(* CODESYS project experiment_with_CoDeSys_sp16.project
   Company: ifm electronic
   Description: Project template with CR711S configured 2.25MByte Standard 2.25MByte Safety
   Version: 2.4.15.0
   Title: ifmCR711S_TemplateProject

Project tree, tasks and I/O mapping:
  SafetyPLC : CR711S SIL2, ifm electronic, order no. CR711S, version 3.0.0.1
    application Application
      libraries: ifmR360-3, * (ifm electronic)
      task Task (cyclic, interval t#10ms, priority 1, watchdog t#8ms x 1) calls PLC_PRG
      global variables EVL
      program PLC_PRG [ST]
    Communication : Communication, ifm electronic, version 3.0.0.1
      CAN : CAN, ifm electronic, version 3.0.0.1
      Ethernet : Ethernet, ifm electronic, version 3.0.0.1
    HMI : HMI, ifm electronic, version 3.0.0.1
      User_LEDs : User_LEDs, ifm electronic, version 3.0.0.1
          input  UserLED0_I : LED_IEC_B_INPUT_MAPPING_TYPE  // UserLED0_I
          input  UserLED1_I : LED_IEC_B_INPUT_MAPPING_TYPE  // UserLED1_I
          input  UserLED2_I : LED_IEC_B_INPUT_MAPPING_TYPE  // UserLED2_I
          input  UserLED3_I : LED_IEC_B_INPUT_MAPPING_TYPE  // UserLED3_I
          output UserLED0_Q : LED_IEC_B_OUTPUT_MAPPING_TYPE  // User LED 0
          output UserLED1_Q : LED_IEC_B_OUTPUT_MAPPING_TYPE  // User LED 1
          output UserLED2_Q : LED_IEC_B_OUTPUT_MAPPING_TYPE  // User LED 2
          output UserLED3_Q : LED_IEC_B_OUTPUT_MAPPING_TYPE  // User LED 3
    Local_IO : Local_IO, ifm electronic, version 3.0.0.1
      Inputs : Inputs, ifm electronic, version 3.0.0.1
          input  IN0100_I : IN_MULTIFUNCTION_A_INPUT_MAPPING_TYPE  // IN0100_I
          input  IN0101_I : IN_MULTIFUNCTION_A_INPUT_MAPPING_TYPE  // IN0101_I
          input  IN0102_I : IN_MULTIFUNCTION_A_INPUT_MAPPING_TYPE  // IN0102_I
          input  IN0103_I : IN_MULTIFUNCTION_A_INPUT_MAPPING_TYPE  // IN0103_I
          input  IN0200_I : IN_MULTIFUNCTION_A_INPUT_MAPPING_TYPE  // IN0200_I
          input  IN0201_I : IN_MULTIFUNCTION_A_INPUT_MAPPING_TYPE  // IN0201_I
          input  IN0202_I : IN_MULTIFUNCTION_A_INPUT_MAPPING_TYPE  // IN0202_I
          input  IN0203_I : IN_MULTIFUNCTION_A_INPUT_MAPPING_TYPE  // IN0203_I
          input  IN0600_I : IN_MULTIFUNCTION_A_INPUT_MAPPING_TYPE  // IN0600_I
          input  IN0601_I : IN_MULTIFUNCTION_A_INPUT_MAPPING_TYPE  // IN0601_I
          input  IN0602_I : IN_MULTIFUNCTION_A_INPUT_MAPPING_TYPE  // IN0602_I
          input  IN0603_I : IN_MULTIFUNCTION_A_INPUT_MAPPING_TYPE  // IN0603_I
          input  IN0700_I : IN_MULTIFUNCTION_A_INPUT_MAPPING_TYPE  // IN0700_I
          input  IN0701_I : IN_MULTIFUNCTION_A_INPUT_MAPPING_TYPE  // IN0701_I
          input  IN0702_I : IN_MULTIFUNCTION_A_INPUT_MAPPING_TYPE  // IN0702_I
          input  IN0703_I : IN_MULTIFUNCTION_A_INPUT_MAPPING_TYPE  // IN0703_I
          input  IN0400_I : IN_RESISTOR_A_INPUT_MAPPING_TYPE  // IN0400_I
          input  IN0401_I : IN_RESISTOR_A_INPUT_MAPPING_TYPE  // IN0401_I
          input  IN0900_I : IN_RESISTOR_A_INPUT_MAPPING_TYPE  // IN0900_I
          input  IN0901_I : IN_RESISTOR_A_INPUT_MAPPING_TYPE  // IN0901_I
          input  IN0300_I : IN_DIGITAL_B_INPUT_MAPPING_TYPE  // IN0300_I
          input  IN0301_I : IN_DIGITAL_B_INPUT_MAPPING_TYPE  // IN0301_I
          input  IN0800_I : IN_DIGITAL_B_INPUT_MAPPING_TYPE  // IN0800_I
          input  IN0801_I : IN_DIGITAL_B_INPUT_MAPPING_TYPE  // IN0801_I
          input  COM_RESET_I : IN_COMMUNICATION_RESET_INPUT_MAPPING_TYPE  // COM_RESET_I
          input  IN0000_I : IN_FREQUENCY_B_CHANNEL_A_INPUT_MAPPING_TYPE  // IN0000_I
          input  IN0002_I : IN_FREQUENCY_B_CHANNEL_A_INPUT_MAPPING_TYPE  // IN0002_I
          input  IN0500_I : IN_FREQUENCY_B_CHANNEL_A_INPUT_MAPPING_TYPE  // IN0500_I
          input  IN0502_I : IN_FREQUENCY_B_CHANNEL_A_INPUT_MAPPING_TYPE  // IN0502_I
          input  IN0001_I : IN_FREQUENCY_B_CHANNEL_B_INPUT_MAPPING_TYPE  // IN0001_I
          input  IN0003_I : IN_FREQUENCY_B_CHANNEL_B_INPUT_MAPPING_TYPE  // IN0003_I
          input  IN0501_I : IN_FREQUENCY_B_CHANNEL_B_INPUT_MAPPING_TYPE  // IN0501_I
          input  IN0503_I : IN_FREQUENCY_B_CHANNEL_B_INPUT_MAPPING_TYPE  // IN0503_I
      Outputs : Outputs, ifm electronic, version 3.0.0.1
          input  OUT0006_I : OUT_PWM_40_BRIDGE_A_INPUT_MAPPING_TYPE  // OUT0006_I
          input  OUT0106_I : OUT_PWM_40_BRIDGE_A_INPUT_MAPPING_TYPE  // OUT0106_I
          input  OUT0206_I : OUT_PWM_40_BRIDGE_A_INPUT_MAPPING_TYPE  // OUT0206_I
          input  OUT0008_I : OUT_PWM_40_A_INPUT_MAPPING_TYPE  // OUT0008_I
          input  OUT0108_I : OUT_PWM_40_A_INPUT_MAPPING_TYPE  // OUT0108_I
          input  OUT0208_I : OUT_PWM_40_A_INPUT_MAPPING_TYPE  // OUT0208_I
          input  OUT0000_I : OUT_PWM_25_A_INPUT_MAPPING_TYPE  // OUT0000_I
          input  OUT0002_I : OUT_PWM_25_A_INPUT_MAPPING_TYPE  // OUT0002_I
          input  OUT0004_I : OUT_PWM_25_A_INPUT_MAPPING_TYPE  // OUT0004_I
          input  OUT0100_I : OUT_PWM_25_A_INPUT_MAPPING_TYPE  // OUT0100_I
          input  OUT0102_I : OUT_PWM_25_A_INPUT_MAPPING_TYPE  // OUT0102_I
          input  OUT0104_I : OUT_PWM_25_A_INPUT_MAPPING_TYPE  // OUT0104_I
          input  OUT0200_I : OUT_PWM_25_A_INPUT_MAPPING_TYPE  // OUT0200_I
          input  OUT0202_I : OUT_PWM_25_A_INPUT_MAPPING_TYPE  // OUT0202_I
          input  OUT0204_I : OUT_PWM_25_A_INPUT_MAPPING_TYPE  // OUT0204_I
          input  OUT3001_I : OUT_VOLTAGE_A_INPUT_MAPPING_TYPE  // OUT3001_I
          input  OUT3000_I : OUT_SUPPLY_A_INPUT_MAPPING_TYPE  // OUT3000_I
          input  OUT0001_I : OUT_PWM_25_B_INPUT_MAPPING_TYPE  // OUT0001_I
          input  OUT0003_I : OUT_PWM_25_B_INPUT_MAPPING_TYPE  // OUT0003_I
          input  OUT0005_I : OUT_PWM_25_B_INPUT_MAPPING_TYPE  // OUT0005_I
          input  OUT0101_I : OUT_PWM_25_B_INPUT_MAPPING_TYPE  // OUT0101_I
          input  OUT0103_I : OUT_PWM_25_B_INPUT_MAPPING_TYPE  // OUT0103_I
          input  OUT0105_I : OUT_PWM_25_B_INPUT_MAPPING_TYPE  // OUT0105_I
          input  OUT0201_I : OUT_PWM_25_B_INPUT_MAPPING_TYPE  // OUT0201_I
          input  OUT0203_I : OUT_PWM_25_B_INPUT_MAPPING_TYPE  // OUT0203_I
          input  OUT0205_I : OUT_PWM_25_B_INPUT_MAPPING_TYPE  // OUT0205_I
          input  OUT0007_I : OUT_PWM_40_BRIDGE_A_INPUT_MAPPING_TYPE  // OUT0007_I
          input  OUT0107_I : OUT_PWM_40_BRIDGE_A_INPUT_MAPPING_TYPE  // OUT0107_I
          input  OUT0207_I : OUT_PWM_40_BRIDGE_A_INPUT_MAPPING_TYPE  // OUT0207_I
          output OUT0006_Q : OUT_PWM_40_BRIDGE_A_OUTPUT_MAPPING_TYPE  // OUT0006_Q
          output OUT0106_Q : OUT_PWM_40_BRIDGE_A_OUTPUT_MAPPING_TYPE  // OUT0106_Q
          output OUT0206_Q : OUT_PWM_40_BRIDGE_A_OUTPUT_MAPPING_TYPE  // OUT0206_Q
          output OUT0008_Q : OUT_PWM_40_A_OUTPUT_MAPPING_TYPE  // OUT0008_Q
          output OUT0108_Q : OUT_PWM_40_A_OUTPUT_MAPPING_TYPE  // OUT0108_Q
          output OUT0208_Q : OUT_PWM_40_A_OUTPUT_MAPPING_TYPE  // OUT0208_Q
          output OUT0000_Q : OUT_PWM_25_A_OUTPUT_MAPPING_TYPE  // OUT0000_Q
          output OUT0002_Q : OUT_PWM_25_A_OUTPUT_MAPPING_TYPE  // OUT0002_Q
          output OUT0004_Q : OUT_PWM_25_A_OUTPUT_MAPPING_TYPE  // OUT0004_Q
          output OUT0100_Q : OUT_PWM_25_A_OUTPUT_MAPPING_TYPE  // OUT0100_Q
          output OUT0102_Q : OUT_PWM_25_A_OUTPUT_MAPPING_TYPE  // OUT0102_Q
          output OUT0104_Q : OUT_PWM_25_A_OUTPUT_MAPPING_TYPE  // OUT0104_Q
          output OUT0200_Q : OUT_PWM_25_A_OUTPUT_MAPPING_TYPE  // OUT0200_Q
          output OUT0202_Q : OUT_PWM_25_A_OUTPUT_MAPPING_TYPE  // OUT0202_Q
          output OUT0204_Q : OUT_PWM_25_A_OUTPUT_MAPPING_TYPE  // OUT0204_Q
          output OUT3001_Q : OUT_VOLTAGE_A_OUTPUT_MAPPING_TYPE  // OUT3001_Q
          output OUT3000_Q : OUT_SUPPLY_A_OUTPUT_MAPPING_TYPE  // OUT3000_Q
          output OUT0001_Q : OUT_PWM_25_B_OUTPUT_MAPPING_TYPE  // OUT0001_Q
          output OUT0003_Q : OUT_PWM_25_B_OUTPUT_MAPPING_TYPE  // OUT0003_Q
          output OUT0005_Q : OUT_PWM_25_B_OUTPUT_MAPPING_TYPE  // OUT0005_Q
          output OUT0101_Q : OUT_PWM_25_B_OUTPUT_MAPPING_TYPE  // OUT0101_Q
          output OUT0103_Q : OUT_PWM_25_B_OUTPUT_MAPPING_TYPE  // OUT0103_Q
          output OUT0105_Q : OUT_PWM_25_B_OUTPUT_MAPPING_TYPE  // OUT0105_Q
          output OUT0201_Q : OUT_PWM_25_B_OUTPUT_MAPPING_TYPE  // OUT0201_Q
          output OUT0203_Q : OUT_PWM_25_B_OUTPUT_MAPPING_TYPE  // OUT0203_Q
          output OUT0205_Q : OUT_PWM_25_B_OUTPUT_MAPPING_TYPE  // OUT0205_Q
          output OUT0007_Q : OUT_PWM_40_BRIDGE_A_OUTPUT_MAPPING_TYPE  // OUT0007_Q
          output OUT0107_Q : OUT_PWM_40_BRIDGE_A_OUTPUT_MAPPING_TYPE  // OUT0107_Q
          output OUT0207_Q : OUT_PWM_40_BRIDGE_A_OUTPUT_MAPPING_TYPE  // OUT0207_Q
      System_Inputs : System_Inputs, ifm electronic, version 3.0.0.1
          input  VBB30 : IN_SYSTEM_VOLTAGE_INPUT_MAPPING_TYPE  // VBB30
          input  VBB15 : IN_SYSTEM_VOLTAGE_INPUT_MAPPING_TYPE  // VBB15
          input  TemperatureBoard0 : IN_TEMPERATURE_INPUT_MAPPING_TYPE  // TemperatureBoard0
          input  TemperatureChip0 : IN_TEMPERATURE_INPUT_MAPPING_TYPE  // TemperatureChip0
      System_Outputs : System_Outputs, ifm electronic, version 3.0.0.1
          input  VBB0_SW_I : OUT_GROUP_SWITCH_INPUT_MAPPING_TYPE  // VBB0_SW_I
          input  VBB1_SW_I : OUT_GROUP_SWITCH_INPUT_MAPPING_TYPE  // VBB1_SW_I
          input  VBB2_SW_I : OUT_GROUP_SWITCH_INPUT_MAPPING_TYPE  // VBB2_SW_I
          output VBB0_SW_Q : OUT_GROUP_SWITCH_OUTPUT_MAPPING_TYPE  // VBB0_SW_Q
          output VBB1_SW_Q : OUT_GROUP_SWITCH_OUTPUT_MAPPING_TYPE  // VBB1_SW_Q
          output VBB2_SW_Q : OUT_GROUP_SWITCH_OUTPUT_MAPPING_TYPE  // VBB2_SW_Q
          output SUPPLY_SWITCH_Q : OUT_SYS_SWITCH_OUTPUT_MAPPING_TYPE  // SUPPLY_SWITCH_Q
  StandardPLC : CR711S Standard, ifm electronic, order no. CR711S, version 3.0.0.1
    application Application
      libraries: ifmR360-3, * (ifm electronic); SysTime, 3.5.9.0 (System); 3S CANopenStack, 3.5.11.0 (3S - Smart Software Solutions GmbH); CAA CiA 405, 3.5.8.0 (CAA Technical Workgroup); Converted Hydraulic library, 0.0.0.1 (ifmWT); StringUtils, 3.5.15.0 (System); SysCom, 3.5.15.0 (System); SysMem23, 3.5.13.0 (System); TD3-1 Framework, 3.1.0.1 (Ojjo); Util, * (System); Motor3-1 control, 3.1.0.1 (Ojjo); Standard, * (System); VisuDialogs, * (System)
      task Task (cyclic, interval 20 ms, priority 1) calls PLC_PRG
      EVC
      GlobalVars/
        global variables Test1Vars
        global variables Test2Vars
        global variables Dims
        global variables Positions
        global variables GPS_Data
        global variables Ojjo_TD
      POUs/
        program PLC_PRG [ST]
        function block ConvertDiag [ST]
        function ConvDiag [ST]
        program Type_conversions [ST]
        function Checksum [ST]
        function Checksum_wLength [ST]
        function IsExtendedCAN [ST]
        function block getElapsedTime [ST]
        Utilities/
          function MemBlockLength [ST]
          Conversions/
            function pSQR [ST]
            function SqrReals [ST]
            function AsciiToReal [ST]
            function ArrayOfBytesToLWORD [ST]
            function ConvLWORDtoDecimal [ST]
            function block REAL_TO_BYTE_ARRAY [ST]
            function ArrayOfUsintsToLWORD [ST]
            function ATAN_DEG [ST]
            function COS_DEG [ST]
            function SIN_DEG [ST]
            function TAN_DEG [ST]
            function CanMsgIdToNodeIndexSubIndex [ST]
            function CanNodeIndexSubIndexToJ1939MsgId [ST]
            function ACOS_DEG [ST]
            function ASIN_DEG [ST]
            function ByteArrayToText [ST]
            function ddt [ST]
            function ddt_max [ST]
            function block ddt_layers [ST]
          ProfileGen/
            function ProfileGenerator_2d [ST]
            function CurveGenerator_2d [ST]
            data type CurveTypes
            function SetpointInit [ST]
            TDcontrolCode/
              function setVelAccel [ST]
              data type sSetpoint
              function POS_ENGR_TO_RAW [ST]
              data type sFeedback
              function FeedbackInit [ST]
              function VEL_ENGR_TO_RAW [ST]
            function block ScurveProfiler [ST]
            function AutotargetIncrementPos [ST]
            function GpsFeedbackAutotarget [ST]
            function TrapezoidStart [ST]
            function TrapezoidStart_jerk [ST]
          function block DataSmoothing [ST]
          function block DataSmoothing_1 [ST]
          function block DataSmoothing_2 [ST]
          function UpperBoundBool [ST]
        GPS/
          data type eScrewParameters
          function RotateGpsTdToWorldNS [ST]
          data type eGPS
          data type eGpsDataCategories
          function GpsTdToWorldFixedYaw [ST]
          function GPS_Y_TO_BS_ANGLE [ST]
          function GPS_Y_TO_BS_ANGLE_1 [ST]
          function GPS_Y_TO_BS_ANGLE_2 [ST]
          function GpsTransform3d [ST]
          function GpsAutotargetInRange [ST]
          data type sGPSaxis
          function block GpsUpdate [ST]
          function block GPS [ST]
          program CheckGpsInRange [ST]
          function TD_SIM [ST]
          function GpsTdToWorldFixAll2d [ST]
          program GpsAutoTrack_1 [ST]
          function GpsAutoTrack [ST]
          function GpsAxisIsNearTarget [ST]
          function GpsAxisIsOnTarget [ST]
          function DecodePnezD [ST]
        Test_PRGs/
          program pnezD_decoding [ST]
          program DynamicList [ST]
          program Arrays [ST]
          program Parsing [ST]
      Network Variables/
        global variables PLC_TRANSMIT_1
      DUTs/
        data type color
        data type SqrStruct
        data type Diag
        data type Coordinates2d
        data type Coordinates3d
        data type sScrewParams
      Visualizations/
        visualisation GPS_RANGE
        visualisation FUNCTION_CHECK
        visualisation P_GPS_testing
        visualisation GRAPH_FUNCTION_RESULTS
    Communication : Communication, ifm electronic, version 3.0.0.1
      CAN : CAN, ifm electronic, version 3.0.0.1
        CANbus_3 : CANbus, ifm electronic, version 1.0.0.0
            settings: NetID = 3
          J1939_Manager : J1939_Manager, 3S - Smart Software Solutions GmbH, version 3.5.10.0
            Rx_KARTECH : J1939_ECU, 3S - Smart Software Solutions GmbH, version 3.5.9.0
                settings: NAME = 16#1060000000000000; Communication Watchdog Timeout Period = 16#05DC ms; Activated PGs = 0; PG Offline Data.Name = "Group0"; PG Offline Data.Description = ""; PG Online Data.PGN = 65280; PG Online Data.Length (Bytes) = 8; PG Transmission Settings.Destination Address = 255; PG Transmission Settings.CycleTimeFactor = 1; Signal Offline Data.SPN = 0; Signal Offline Data.Name = "Toggle"; Signal Offline Data.Description = ""; Signal Offline Data.Unit = ""; Signal Offline Data.Min = 0; Signal Offline Data.Max = 0; Signal Online Data.BitSize = 1; Signal Online Data.BitPosition = 0; Convert Data.Flags = 3; Convert Data.pSigValue = 0; Convert Data.Scaling = 4607182418800017408; Convert Data.Offset = 0; Signal Offline Data.SPN = 0; Signal Offline Data.Name = "rf_CANlink"; Signal Offline Data.Description = ""; Signal Offline Data.Unit = ""; Signal Offline Data.Min = 0; Signal Offline Data.Max = 0; Signal Online Data.BitSize = 1; Signal Online Data.BitPosition = 1; Convert Data.Flags = 3; Convert Data.pSigValue = 0; Convert Data.Scaling = 4607182418800017408; Convert Data.Offset = 0; Signal Offline Data.SPN = 0; Signal Offline Data.Name = "DI1"; Signal Offline Data.Description = ""; Signal Offline Data.Unit = ""; Signal Offline Data.Min = 0; Signal Offline Data.Max = 0; Signal Online Data.BitSize = 1;
                  Signal Online Data.BitPosition = 16; Convert Data.Flags = 3; Convert Data.pSigValue = 0; Convert Data.Scaling = 4607182418800017408; Convert Data.Offset = 0; Signal Offline Data.SPN = 0; Signal Offline Data.Name = "DI2"; Signal Offline Data.Description = ""; Signal Offline Data.Unit = ""; Signal Offline Data.Min = 0; Signal Offline Data.Max = 0; Signal Online Data.BitSize = 1; Signal Online Data.BitPosition = 17; Convert Data.Flags = 3; Convert Data.pSigValue = 0; Convert Data.Scaling = 4607182418800017408; Convert Data.Offset = 0; Signal Offline Data.SPN = 0; Signal Offline Data.Name = "DI3"; Signal Offline Data.Description = ""; Signal Offline Data.Unit = ""; Signal Offline Data.Min = 0; Signal Offline Data.Max = 0; Signal Online Data.BitSize = 1; Signal Online Data.BitPosition = 18; Convert Data.Flags = 3; Convert Data.pSigValue = 0; Convert Data.Scaling = 4607182418800017408; Convert Data.Offset = 0; Signal Offline Data.SPN = 0; Signal Offline Data.Name = "DI4"; Signal Offline Data.Description = ""; Signal Offline Data.Unit = ""; Signal Offline Data.Min = 0; Signal Offline Data.Max = 0; Signal Online Data.BitSize = 1; Signal Online Data.BitPosition = 19; Convert Data.Flags = 3; Convert Data.pSigValue = 0; Convert Data.Scaling = 4607182418800017408;
                  Convert Data.Offset = 0; Signal Offline Data.SPN = 0; Signal Offline Data.Name = "DI5"; Signal Offline Data.Description = ""; Signal Offline Data.Unit = ""; Signal Offline Data.Min = 0; Signal Offline Data.Max = 0; Signal Online Data.BitSize = 1; Signal Online Data.BitPosition = 20; Convert Data.Flags = 3; Convert Data.pSigValue = 0; Convert Data.Scaling = 4607182418800017408; Convert Data.Offset = 0; Signal Offline Data.SPN = 0; Signal Offline Data.Name = "DI6"; Signal Offline Data.Description = ""; Signal Offline Data.Unit = ""; Signal Offline Data.Min = 0; Signal Offline Data.Max = 0; Signal Online Data.BitSize = 1; Signal Online Data.BitPosition = 21; Convert Data.Flags = 3; Convert Data.pSigValue = 0; Convert Data.Scaling = 4607182418800017408; Convert Data.Offset = 0; Signal Offline Data.SPN = 0; Signal Offline Data.Name = "DI7"; Signal Offline Data.Description = ""; Signal Offline Data.Unit = ""; Signal Offline Data.Min = 0; Signal Offline Data.Max = 0; Signal Online Data.BitSize = 1; Signal Online Data.BitPosition = 22; Convert Data.Flags = 3; Convert Data.pSigValue = 0; Convert Data.Scaling = 4607182418800017408; Convert Data.Offset = 0; Signal Offline Data.SPN = 0; Signal Offline Data.Name = "DI8"; Signal Offline Data.Description = "";
                  Signal Offline Data.Unit = ""; Signal Offline Data.Min = 0; Signal Offline Data.Max = 0; Signal Online Data.BitSize = 1; Signal Online Data.BitPosition = 23; Convert Data.Flags = 3; Convert Data.pSigValue = 0; Convert Data.Scaling = 4607182418800017408; Convert Data.Offset = 0; Signal Offline Data.SPN = 0; Signal Offline Data.Name = "DI9"; Signal Offline Data.Description = ""; Signal Offline Data.Unit = ""; Signal Offline Data.Min = 0; Signal Offline Data.Max = 0; Signal Online Data.BitSize = 1; Signal Online Data.BitPosition = 24; Convert Data.Flags = 3; Convert Data.pSigValue = 0; Convert Data.Scaling = 4607182418800017408; Convert Data.Offset = 0; Signal Offline Data.SPN = 0; Signal Offline Data.Name = "DI10"; Signal Offline Data.Description = ""; Signal Offline Data.Unit = ""; Signal Offline Data.Min = 0; Signal Offline Data.Max = 0; Signal Online Data.BitSize = 1; Signal Online Data.BitPosition = 25; Convert Data.Flags = 3; Convert Data.pSigValue = 0; Convert Data.Scaling = 4607182418800017408; Convert Data.Offset = 0; Signal Offline Data.SPN = 0; Signal Offline Data.Name = "DI11"; Signal Offline Data.Description = ""; Signal Offline Data.Unit = ""; Signal Offline Data.Min = 0; Signal Offline Data.Max = 0; Signal Online Data.BitSize = 1;
                  Signal Online Data.BitPosition = 26; Convert Data.Flags = 3; Convert Data.pSigValue = 0; Convert Data.Scaling = 4607182418800017408; Convert Data.Offset = 0; Signal Offline Data.SPN = 0; Signal Offline Data.Name = "DI12"; Signal Offline Data.Description = ""; Signal Offline Data.Unit = ""; Signal Offline Data.Min = 0; Signal Offline Data.Max = 0; Signal Online Data.BitSize = 1; Signal Online Data.BitPosition = 27; Convert Data.Flags = 3; Convert Data.pSigValue = 0; Convert Data.Scaling = 4607182418800017408; Convert Data.Offset = 0; Signal Offline Data.SPN = 0; Signal Offline Data.Name = "DI13"; Signal Offline Data.Description = ""; Signal Offline Data.Unit = ""; Signal Offline Data.Min = 0; Signal Offline Data.Max = 0; Signal Online Data.BitSize = 1; Signal Online Data.BitPosition = 28; Convert Data.Flags = 3; Convert Data.pSigValue = 0; Convert Data.Scaling = 4607182418800017408; Convert Data.Offset = 0; Signal Offline Data.SPN = 0; Signal Offline Data.Name = "DI14"; Signal Offline Data.Description = ""; Signal Offline Data.Unit = ""; Signal Offline Data.Min = 0; Signal Offline Data.Max = 0; Signal Online Data.BitSize = 1; Signal Online Data.BitPosition = 29; Convert Data.Flags = 3; Convert Data.pSigValue = 0; Convert Data.Scaling = 4607182418800017408;
                  Convert Data.Offset = 0; Signal Offline Data.SPN = 0; Signal Offline Data.Name = "DI15"; Signal Offline Data.Description = ""; Signal Offline Data.Unit = ""; Signal Offline Data.Min = 0; Signal Offline Data.Max = 0; Signal Online Data.BitSize = 1; Signal Online Data.BitPosition = 30; Convert Data.Flags = 3; Convert Data.pSigValue = 0; Convert Data.Scaling = 4607182418800017408; Convert Data.Offset = 0; Signal Offline Data.SPN = 0; Signal Offline Data.Name = "DI16"; Signal Offline Data.Description = ""; Signal Offline Data.Unit = ""; Signal Offline Data.Min = 0; Signal Offline Data.Max = 0; Signal Online Data.BitSize = 1; Signal Online Data.BitPosition = 31; Convert Data.Flags = 3; Convert Data.pSigValue = 0; Convert Data.Scaling = 4607182418800017408; Convert Data.Offset = 0; Signal Offline Data.SPN = 0; Signal Offline Data.Name = "DI17"; Signal Offline Data.Description = ""; Signal Offline Data.Unit = ""; Signal Offline Data.Min = 0; Signal Offline Data.Max = 0; Signal Online Data.BitSize = 1; Signal Online Data.BitPosition = 32; Convert Data.Flags = 3; Convert Data.pSigValue = 0; Convert Data.Scaling = 4607182418800017408; Convert Data.Offset = 0; Signal Offline Data.SPN = 0; Signal Offline Data.Name = "DI18"; Signal Offline Data.Description = "";
                  Signal Offline Data.Unit = ""; Signal Offline Data.Min = 0; Signal Offline Data.Max = 0; Signal Online Data.BitSize = 1; Signal Online Data.BitPosition = 33; Convert Data.Flags = 3; Convert Data.pSigValue = 0; Convert Data.Scaling = 4607182418800017408; Convert Data.Offset = 0; Signal Offline Data.SPN = 0; Signal Offline Data.Name = "DI19"; Signal Offline Data.Description = ""; Signal Offline Data.Unit = ""; Signal Offline Data.Min = 0; Signal Offline Data.Max = 0; Signal Online Data.BitSize = 1; Signal Online Data.BitPosition = 34; Convert Data.Flags = 3; Convert Data.pSigValue = 0; Convert Data.Scaling = 4607182418800017408; Convert Data.Offset = 0; Signal Offline Data.SPN = 0; Signal Offline Data.Name = "DI20"; Signal Offline Data.Description = ""; Signal Offline Data.Unit = ""; Signal Offline Data.Min = 0; Signal Offline Data.Max = 0; Signal Online Data.BitSize = 1; Signal Online Data.BitPosition = 35; Convert Data.Flags = 3; Convert Data.pSigValue = 0; Convert Data.Scaling = 4607182418800017408; Convert Data.Offset = 0; PG Offline Data.Name = "Group1"; PG Offline Data.Description = ""; PG Online Data.PGN = 65281; PG Online Data.Length (Bytes) = 8; PG Transmission Settings.Destination Address = 255; PG Transmission Settings.CycleTimeFactor = 1; Signal Offline Data.SPN = 0;
                  Signal Offline Data.Name = "AI1"; Signal Offline Data.Description = ""; Signal Offline Data.Unit = ""; Signal Offline Data.Min = 0; Signal Offline Data.Max = 0; Signal Online Data.BitSize = 8; Signal Online Data.BitPosition = 0; Convert Data.Flags = 3; Convert Data.pSigValue = 0; Convert Data.Scaling = 4607182418800017408; Convert Data.Offset = 0; Signal Offline Data.SPN = 0; Signal Offline Data.Name = "AI2"; Signal Offline Data.Description = ""; Signal Offline Data.Unit = ""; Signal Offline Data.Min = 0; Signal Offline Data.Max = 0; Signal Online Data.BitSize = 8; Signal Online Data.BitPosition = 8; Convert Data.Flags = 3; Convert Data.pSigValue = 0; Convert Data.Scaling = 4607182418800017408; Convert Data.Offset = 0; Signal Offline Data.SPN = 0; Signal Offline Data.Name = "AI3"; Signal Offline Data.Description = ""; Signal Offline Data.Unit = ""; Signal Offline Data.Min = 0; Signal Offline Data.Max = 0; Signal Online Data.BitSize = 8; Signal Online Data.BitPosition = 16; Convert Data.Flags = 3; Convert Data.pSigValue = 0; Convert Data.Scaling = 4607182418800017408; Convert Data.Offset = 0; Signal Offline Data.SPN = 0; Signal Offline Data.Name = "AI4"; Signal Offline Data.Description = ""; Signal Offline Data.Unit = ""; Signal Offline Data.Min = 0;
                  Signal Offline Data.Max = 0; Signal Online Data.BitSize = 8; Signal Online Data.BitPosition = 24; Convert Data.Flags = 3; Convert Data.pSigValue = 0; Convert Data.Scaling = 4607182418800017408; Convert Data.Offset = 0; Signal Offline Data.SPN = 0; Signal Offline Data.Name = "AI5"; Signal Offline Data.Description = ""; Signal Offline Data.Unit = ""; Signal Offline Data.Min = 0; Signal Offline Data.Max = 0; Signal Online Data.BitSize = 8; Signal Online Data.BitPosition = 32; Convert Data.Flags = 3; Convert Data.pSigValue = 0; Convert Data.Scaling = 4607182418800017408; Convert Data.Offset = 0; Signal Offline Data.SPN = 0; Signal Offline Data.Name = "AI6"; Signal Offline Data.Description = ""; Signal Offline Data.Unit = ""; Signal Offline Data.Min = 0; Signal Offline Data.Max = 0; Signal Online Data.BitSize = 8; Signal Online Data.BitPosition = 40; Convert Data.Flags = 3; Convert Data.pSigValue = 0; Convert Data.Scaling = 4607182418800017408; Convert Data.Offset = 0; Signal Offline Data.SPN = 0; Signal Offline Data.Name = "AI7"; Signal Offline Data.Description = ""; Signal Offline Data.Unit = ""; Signal Offline Data.Min = 0; Signal Offline Data.Max = 0; Signal Online Data.BitSize = 8; Signal Online Data.BitPosition = 48; Convert Data.Flags = 3;
                  Convert Data.pSigValue = 0; Convert Data.Scaling = 4607182418800017408; Convert Data.Offset = 0; Signal Offline Data.SPN = 0; Signal Offline Data.Name = "AI8"; Signal Offline Data.Description = ""; Signal Offline Data.Unit = ""; Signal Offline Data.Min = 0; Signal Offline Data.Max = 0; Signal Online Data.BitSize = 8; Signal Online Data.BitPosition = 56; Convert Data.Flags = 3; Convert Data.pSigValue = 0; Convert Data.Scaling = 4607182418800017408; Convert Data.Offset = 0; PG Offline Data.Name = "Group2"; PG Offline Data.Description = ""; PG Online Data.PGN = 65282; PG Online Data.Length (Bytes) = 8; PG Transmission Settings.Destination Address = 255; PG Transmission Settings.CycleTimeFactor = 1; Signal Offline Data.SPN = 0; Signal Offline Data.Name = "BatteryVoltage"; Signal Offline Data.Description = ""; Signal Offline Data.Unit = ""; Signal Offline Data.Min = 0; Signal Offline Data.Max = 0; Signal Online Data.BitSize = 16; Signal Online Data.BitPosition = 0; Convert Data.Flags = 3; Convert Data.pSigValue = 0; Convert Data.Scaling = 4607182418800017408; Convert Data.Offset = 4587366580439587226; Signal Offline Data.SPN = 0; Signal Offline Data.Name = "low_voltage"; Signal Offline Data.Description = ""; Signal Offline Data.Unit = ""; Signal Offline Data.Min = 0; Signal Offline Data.Max = 0; Signal Online Data.BitSize = 1;
                  Signal Online Data.BitPosition = 16; Convert Data.Flags = 3; Convert Data.pSigValue = 0; Convert Data.Scaling = 4607182418800017408; Convert Data.Offset = 0; Signal Offline Data.SPN = 0; Signal Offline Data.Name = "aiInput1err"; Signal Offline Data.Description = ""; Signal Offline Data.Unit = ""; Signal Offline Data.Min = 0; Signal Offline Data.Max = 0; Signal Online Data.BitSize = 1; Signal Online Data.BitPosition = 17; Convert Data.Flags = 3; Convert Data.pSigValue = 0; Convert Data.Scaling = 4607182418800017408; Convert Data.Offset = 0; Signal Offline Data.SPN = 0; Signal Offline Data.Name = "aiInput2err"; Signal Offline Data.Description = ""; Signal Offline Data.Unit = ""; Signal Offline Data.Min = 0; Signal Offline Data.Max = 0; Signal Online Data.BitSize = 1; Signal Online Data.BitPosition = 18; Convert Data.Flags = 3; Convert Data.pSigValue = 0; Convert Data.Scaling = 4607182418800017408; Convert Data.Offset = 0; Signal Offline Data.SPN = 0; Signal Offline Data.Name = "aiInput3err"; Signal Offline Data.Description = ""; Signal Offline Data.Unit = ""; Signal Offline Data.Min = 0; Signal Offline Data.Max = 0; Signal Online Data.BitSize = 1; Signal Online Data.BitPosition = 19; Convert Data.Flags = 3; Convert Data.pSigValue = 0; Convert Data.Scaling = 4607182418800017408;
                  Convert Data.Offset = 0; Signal Offline Data.SPN = 0; Signal Offline Data.Name = "aiInput4err"; Signal Offline Data.Description = ""; Signal Offline Data.Unit = ""; Signal Offline Data.Min = 0; Signal Offline Data.Max = 0; Signal Online Data.BitSize = 1; Signal Online Data.BitPosition = 20; Convert Data.Flags = 3; Convert Data.pSigValue = 0; Convert Data.Scaling = 4607182418800017408; Convert Data.Offset = 0; Signal Offline Data.SPN = 0; Signal Offline Data.Name = "aiInput5err"; Signal Offline Data.Description = ""; Signal Offline Data.Unit = ""; Signal Offline Data.Min = 0; Signal Offline Data.Max = 0; Signal Online Data.BitSize = 1; Signal Online Data.BitPosition = 21; Convert Data.Flags = 3; Convert Data.pSigValue = 0; Convert Data.Scaling = 4607182418800017408; Convert Data.Offset = 0; Signal Offline Data.SPN = 0; Signal Offline Data.Name = "aiInput6err"; Signal Offline Data.Description = ""; Signal Offline Data.Unit = ""; Signal Offline Data.Min = 0; Signal Offline Data.Max = 0; Signal Online Data.BitSize = 1; Signal Online Data.BitPosition = 22; Convert Data.Flags = 3; Convert Data.pSigValue = 0; Convert Data.Scaling = 4607182418800017408; Convert Data.Offset = 0; Signal Offline Data.SPN = 0; Signal Offline Data.Name = "aiInput7err"; Signal Offline Data.Description = "";
                  Signal Offline Data.Unit = ""; Signal Offline Data.Min = 0; Signal Offline Data.Max = 0; Signal Online Data.BitSize = 1; Signal Online Data.BitPosition = 23; Convert Data.Flags = 3; Convert Data.pSigValue = 0; Convert Data.Scaling = 4607182418800017408; Convert Data.Offset = 0; Signal Offline Data.SPN = 0; Signal Offline Data.Name = "aiInput8err"; Signal Offline Data.Description = ""; Signal Offline Data.Unit = ""; Signal Offline Data.Min = 0; Signal Offline Data.Max = 0; Signal Online Data.BitSize = 1; Signal Online Data.BitPosition = 24; Convert Data.Flags = 3; Convert Data.pSigValue = 0; Convert Data.Scaling = 4607182418800017408; Convert Data.Offset = 0; Signal Offline Data.SPN = 0; Signal Offline Data.Name = "VendorID"; Signal Offline Data.Description = ""; Signal Offline Data.Unit = ""; Signal Offline Data.Min = 0; Signal Offline Data.Max = 0; Signal Online Data.BitSize = 7; Signal Online Data.BitPosition = 25; Convert Data.Flags = 3; Convert Data.pSigValue = 0; Convert Data.Scaling = 4607182418800017408; Convert Data.Offset = 0; Signal Offline Data.SPN = 0; Signal Offline Data.Name = "Byte3"; Signal Offline Data.Description = ""; Signal Offline Data.Unit = ""; Signal Offline Data.Min = 0; Signal Offline Data.Max = 0; Signal Online Data.BitSize = 8;
                  Signal Online Data.BitPosition = 32; Convert Data.Flags = 3; Convert Data.pSigValue = 0; Convert Data.Scaling = 4607182418800017408; Convert Data.Offset = 0; Signal Offline Data.SPN = 0; Signal Offline Data.Name = "Byte4"; Signal Offline Data.Description = ""; Signal Offline Data.Unit = ""; Signal Offline Data.Min = 0; Signal Offline Data.Max = 0; Signal Online Data.BitSize = 8; Signal Online Data.BitPosition = 40; Convert Data.Flags = 3; Convert Data.pSigValue = 0; Convert Data.Scaling = 4607182418800017408; Convert Data.Offset = 0; Signal Offline Data.SPN = 0; Signal Offline Data.Name = "Byte5"; Signal Offline Data.Description = ""; Signal Offline Data.Unit = ""; Signal Offline Data.Min = 0; Signal Offline Data.Max = 0; Signal Online Data.BitSize = 8; Signal Online Data.BitPosition = 48; Convert Data.Flags = 3; Convert Data.pSigValue = 0; Convert Data.Scaling = 4607182418800017408; Convert Data.Offset = 0; Signal Offline Data.SPN = 0; Signal Offline Data.Name = "Byte6"; Signal Offline Data.Description = ""; Signal Offline Data.Unit = ""; Signal Offline Data.Min = 0; Signal Offline Data.Max = 0; Signal Online Data.BitSize = 8; Signal Online Data.BitPosition = 56; Convert Data.Flags = 3; Convert Data.pSigValue = 0; Convert Data.Scaling = 4607182418800017408;
                  Convert Data.Offset = 0; Signal Offline Data.SPN = 0; Signal Offline Data.Name = "Byte7"; Signal Offline Data.Description = ""; Signal Offline Data.Unit = ""; Signal Offline Data.Min = 0; Signal Offline Data.Max = 0; Signal Online Data.BitSize = 8; Signal Online Data.BitPosition = 57; Convert Data.Flags = 3; Convert Data.pSigValue = 0; Convert Data.Scaling = 4607182418800017408; Convert Data.Offset = 0; Activated PGs = 0
            LHP_Telematics : J1939_ECU, 3S - Smart Software Solutions GmbH, version 3.5.9.0
                settings: NAME = 16#0000000000000000; Communication Watchdog Timeout Period = 16#05DC ms; Activated PGs = 3; PG Offline Data.Name = "VP"; PG Offline Data.Description = "Vehicle Position"; PG Online Data.PGN = 65267; PG Online Data.Length (Bytes) = 8; PG Transmission Settings.Destination Address = 255; PG Transmission Settings.CycleTimeFactor = 1; Signal Offline Data.SPN = 584; Signal Offline Data.Name = "Latitude"; Signal Offline Data.Description = "Latitude position of the vehicle."; Signal Offline Data.Unit = "deg"; Signal Offline Data.Min = -210; Signal Offline Data.Max = 211.1008122; Signal Online Data.BitSize = 32; Signal Online Data.BitPosition = 0; Convert Data.Flags = 3; Convert Data.pSigValue = 0; Convert Data.Scaling = 4502148214488346440; Convert Data.Offset = 13864964771557670912; Signal Offline Data.SPN = 585; Signal Offline Data.Name = "Longitude"; Signal Offline Data.Description = "Longitude position of the vehicle."; Signal Offline Data.Unit = "deg"; Signal Offline Data.Min = -210; Signal Offline Data.Max = 211.1008122; Signal Online Data.BitSize = 32; Signal Online Data.BitPosition = 32; Convert Data.Flags = 3; Convert Data.pSigValue = 0; Convert Data.Scaling = 4502148214488346440; Convert Data.Offset = 13864964771557670912; PG Offline Data.Name = "VDS"; PG Offline Data.Description = "Vehicle Direction/Speed"; PG Online Data.PGN = 65256; PG Online Data.Length (Bytes) = 8; PG Transmission Settings.Destination Address = 255; PG Transmission Settings.CycleTimeFactor = 1; Signal Offline Data.SPN = 165;
                  Signal Offline Data.Name = "Compass Bearing"; Signal Offline Data.Description = "Present compass bearing of vehicle."; Signal Offline Data.Unit = "deg"; Signal Offline Data.Min = 0; Signal Offline Data.Max = 501.99; Signal Online Data.BitSize = 16; Signal Online Data.BitPosition = 0; Convert Data.Flags = 3; Convert Data.pSigValue = 0; Convert Data.Scaling = 4575657221408423936; Convert Data.Offset = 0; Signal Offline Data.SPN = 517; Signal Offline Data.Name = "Navigation-Based Vehicle Speed"; Signal Offline Data.Description = "Speed of the vehicle as calculated from a device such as a Global Positioning System (GPS)."; Signal Offline Data.Unit = "kph"; Signal Offline Data.Min = 0; Signal Offline Data.Max = 250.996; Signal Online Data.BitSize = 16; Signal Online Data.BitPosition = 16; Convert Data.Flags = 3; Convert Data.pSigValue = 0; Convert Data.Scaling = 4571153621781053440; Convert Data.Offset = 0; Signal Offline Data.SPN = 583; Signal Offline Data.Name = "Pitch"; Signal Offline Data.Unit = "deg"; Signal Offline Data.Min = -200; Signal Offline Data.Max = 301.99; Signal Online Data.BitSize = 16; Signal Online Data.BitPosition = 32; Convert Data.Flags = 3; Convert Data.pSigValue = 0; Convert Data.Scaling = 4575657221408423936; Convert Data.Offset = 13864612927836782592; Signal Offline Data.SPN = 580; Signal Offline Data.Name = "Altitude"; Signal Offline Data.Description = "Altitude of the vehicle referenced to sea level at standard atmospheric pressure and temperature."; Signal Offline Data.Unit = "m"; Signal Offline Data.Min = -2500; Signal Offline Data.Max = 5531.875;
                  Signal Online Data.BitSize = 16; Signal Online Data.BitPosition = 48; Convert Data.Flags = 3; Convert Data.pSigValue = 0; Convert Data.Scaling = 4593671619917905920; Convert Data.Offset = 13881088010067378176; PG Offline Data.Name = "Vehicle Position 2"; PG Offline Data.Description = ""; PG Online Data.PGN = 64502; PG Online Data.Length (Bytes) = 64; PG Transmission Settings.Destination Address = 255; PG Transmission Settings.CycleTimeFactor = 1; Signal Offline Data.SPN = 520; Signal Offline Data.Name = "num_satellites"; Signal Offline Data.Description = ""; Signal Offline Data.Unit = ""; Signal Offline Data.Min = 0; Signal Offline Data.Max = 0; Signal Online Data.BitSize = 8; Signal Online Data.BitPosition = 0; Convert Data.Flags = 3; Convert Data.pSigValue = 0; Convert Data.Scaling = 4607182418800017408; Convert Data.Offset = 0; Signal Offline Data.SPN = 521; Signal Offline Data.Name = "HorizontalDilutionOfPrecision"; Signal Offline Data.Description = ""; Signal Offline Data.Unit = ""; Signal Offline Data.Min = 0; Signal Offline Data.Max = 0; Signal Online Data.BitSize = 8; Signal Online Data.BitPosition = 8; Convert Data.Flags = 3; Convert Data.pSigValue = 0; Convert Data.Scaling = 4607182418800017408; Convert Data.Offset = 0; Signal Offline Data.SPN = 522; Signal Offline Data.Name = "VerticalDilutionOfPrecision"; Signal Offline Data.Description = ""; Signal Offline Data.Unit = "";
                  Signal Offline Data.Min = 0; Signal Offline Data.Max = 0; Signal Online Data.BitSize = 8; Signal Online Data.BitPosition = 16; Convert Data.Flags = 3; Convert Data.pSigValue = 0; Convert Data.Scaling = 4607182418800017408; Convert Data.Offset = 0; Signal Offline Data.SPN = 523; Signal Offline Data.Name = "PositionDilutionOfPrecision"; Signal Offline Data.Description = ""; Signal Offline Data.Unit = ""; Signal Offline Data.Min = 0; Signal Offline Data.Max = 0; Signal Online Data.BitSize = 8; Signal Online Data.BitPosition = 24; Convert Data.Flags = 3; Convert Data.pSigValue = 0; Convert Data.Scaling = 4607182418800017408; Convert Data.Offset = 0; Signal Offline Data.SPN = 524; Signal Offline Data.Name = "TimeDilutionOfPrecision"; Signal Offline Data.Description = ""; Signal Offline Data.Unit = ""; Signal Offline Data.Min = 0; Signal Offline Data.Max = 0; Signal Online Data.BitSize = 8; Signal Online Data.BitPosition = 32; Convert Data.Flags = 3; Convert Data.pSigValue = 0; Convert Data.Scaling = 4607182418800017408; Convert Data.Offset = 0
                input  Latitude_lhp : REAL  // Latitude
                input  Longitude_lhp : REAL  // Longitude
                input  Compass_Bearing : localTypes:TByteArray2  // Compass Bearing
                input  Navigation_Based_Vehicle_Speed : REAL  // Navigation-Based Vehicle Speed
                input  Pitch_lhp : REAL  // Pitch
                input  Altitude_lhp : REAL  // Altitude
                input  num_satellites : BYTE  // num_satellites
                input  HorizontalDilutionOfPrecision_1 : BYTE  // HorizontalDilutionOfPrecision
                input  VerticalDilutionOfPrecision_1 : BYTE  // VerticalDilutionOfPrecision
                input  PositionDilutionOfPrecision_1 : BYTE  // PositionDilutionOfPrecision
                input  TimeDilutionOfPrecision_1 : BYTE  // TimeDilutionOfPrecision
      Ethernet : Ethernet, ifm electronic, version 3.0.0.1
    HMI : HMI, ifm electronic, version 3.0.0.1
      User_LEDs : User_LEDs, ifm electronic, version 3.0.0.1
          input  UserLED0_I : LED_IEC_B_INPUT_MAPPING_TYPE  // UserLED0_I
          input  UserLED1_I : LED_IEC_B_INPUT_MAPPING_TYPE  // UserLED1_I
          input  UserLED2_I : LED_IEC_B_INPUT_MAPPING_TYPE  // UserLED2_I
          input  UserLED3_I : LED_IEC_B_INPUT_MAPPING_TYPE  // UserLED3_I
          output UserLED0_Q : LED_IEC_B_OUTPUT_MAPPING_TYPE  // User LED 0
          output UserLED1_Q : LED_IEC_B_OUTPUT_MAPPING_TYPE  // User LED 1
          output UserLED2_Q : LED_IEC_B_OUTPUT_MAPPING_TYPE  // User LED 2
          output UserLED3_Q : LED_IEC_B_OUTPUT_MAPPING_TYPE  // User LED 3
    Local_IO : Local_IO, ifm electronic, version 3.0.0.1
      Inputs : Inputs, ifm electronic, version 3.0.0.1
          input  IN0100_I : IN_MULTIFUNCTION_A_INPUT_MAPPING_TYPE  // IN0100_I
          input  IN0101_I : IN_MULTIFUNCTION_A_INPUT_MAPPING_TYPE  // IN0101_I
          input  IN0102_I : IN_MULTIFUNCTION_A_INPUT_MAPPING_TYPE  // IN0102_I
          input  IN0103_I : IN_MULTIFUNCTION_A_INPUT_MAPPING_TYPE  // IN0103_I
          input  IN0200_I : IN_MULTIFUNCTION_A_INPUT_MAPPING_TYPE  // IN0200_I
          input  IN0201_I : IN_MULTIFUNCTION_A_INPUT_MAPPING_TYPE  // IN0201_I
          input  IN0202_I : IN_MULTIFUNCTION_A_INPUT_MAPPING_TYPE  // IN0202_I
          input  IN0203_I : IN_MULTIFUNCTION_A_INPUT_MAPPING_TYPE  // IN0203_I
          input  IN0600_I : IN_MULTIFUNCTION_A_INPUT_MAPPING_TYPE  // IN0600_I
          input  IN0601_I : IN_MULTIFUNCTION_A_INPUT_MAPPING_TYPE  // IN0601_I
          input  IN0602_I : IN_MULTIFUNCTION_A_INPUT_MAPPING_TYPE  // IN0602_I
          input  IN0603_I : IN_MULTIFUNCTION_A_INPUT_MAPPING_TYPE  // IN0603_I
          input  IN0700_I : IN_MULTIFUNCTION_A_INPUT_MAPPING_TYPE  // IN0700_I
          input  IN0701_I : IN_MULTIFUNCTION_A_INPUT_MAPPING_TYPE  // IN0701_I
          input  IN0702_I : IN_MULTIFUNCTION_A_INPUT_MAPPING_TYPE  // IN0702_I
          input  IN0703_I : IN_MULTIFUNCTION_A_INPUT_MAPPING_TYPE  // IN0703_I
          input  IN0400_I : IN_RESISTOR_A_INPUT_MAPPING_TYPE  // IN0400_I
          input  IN0401_I : IN_RESISTOR_A_INPUT_MAPPING_TYPE  // IN0401_I
          input  IN0900_I : IN_RESISTOR_A_INPUT_MAPPING_TYPE  // IN0900_I
          input  IN0901_I : IN_RESISTOR_A_INPUT_MAPPING_TYPE  // IN0901_I
          input  IN0300_I : IN_DIGITAL_B_INPUT_MAPPING_TYPE  // IN0300_I
          input  IN0301_I : IN_DIGITAL_B_INPUT_MAPPING_TYPE  // IN0301_I
          input  IN0800_I : IN_DIGITAL_B_INPUT_MAPPING_TYPE  // IN0800_I
          input  IN0801_I : IN_DIGITAL_B_INPUT_MAPPING_TYPE  // IN0801_I
          input  COM_RESET_I : IN_COMMUNICATION_RESET_INPUT_MAPPING_TYPE  // COM_RESET_I
          input  IN0000_I : IN_FREQUENCY_B_CHANNEL_A_INPUT_MAPPING_TYPE  // IN0000_I
          input  IN0002_I : IN_FREQUENCY_B_CHANNEL_A_INPUT_MAPPING_TYPE  // IN0002_I
          input  IN0500_I : IN_FREQUENCY_B_CHANNEL_A_INPUT_MAPPING_TYPE  // IN0500_I
          input  IN0502_I : IN_FREQUENCY_B_CHANNEL_A_INPUT_MAPPING_TYPE  // IN0502_I
          input  IN0001_I : IN_FREQUENCY_B_CHANNEL_B_INPUT_MAPPING_TYPE  // IN0001_I
          input  IN0003_I : IN_FREQUENCY_B_CHANNEL_B_INPUT_MAPPING_TYPE  // IN0003_I
          input  IN0501_I : IN_FREQUENCY_B_CHANNEL_B_INPUT_MAPPING_TYPE  // IN0501_I
          input  IN0503_I : IN_FREQUENCY_B_CHANNEL_B_INPUT_MAPPING_TYPE  // IN0503_I
      Outputs : Outputs, ifm electronic, version 3.0.0.1
          input  OUT0006_I : OUT_PWM_40_BRIDGE_A_INPUT_MAPPING_TYPE  // OUT0006_I
          input  OUT0106_I : OUT_PWM_40_BRIDGE_A_INPUT_MAPPING_TYPE  // OUT0106_I
          input  OUT0206_I : OUT_PWM_40_BRIDGE_A_INPUT_MAPPING_TYPE  // OUT0206_I
          input  OUT0008_I : OUT_PWM_40_A_INPUT_MAPPING_TYPE  // OUT0008_I
          input  OUT0108_I : OUT_PWM_40_A_INPUT_MAPPING_TYPE  // OUT0108_I
          input  OUT0208_I : OUT_PWM_40_A_INPUT_MAPPING_TYPE  // OUT0208_I
          input  OUT0000_I : OUT_PWM_25_A_INPUT_MAPPING_TYPE  // OUT0000_I
          input  OUT0002_I : OUT_PWM_25_A_INPUT_MAPPING_TYPE  // OUT0002_I
          input  OUT0004_I : OUT_PWM_25_A_INPUT_MAPPING_TYPE  // OUT0004_I
          input  OUT0100_I : OUT_PWM_25_A_INPUT_MAPPING_TYPE  // OUT0100_I
          input  OUT0102_I : OUT_PWM_25_A_INPUT_MAPPING_TYPE  // OUT0102_I
          input  OUT0104_I : OUT_PWM_25_A_INPUT_MAPPING_TYPE  // OUT0104_I
          input  OUT0200_I : OUT_PWM_25_A_INPUT_MAPPING_TYPE  // OUT0200_I
          input  OUT0202_I : OUT_PWM_25_A_INPUT_MAPPING_TYPE  // OUT0202_I
          input  OUT0204_I : OUT_PWM_25_A_INPUT_MAPPING_TYPE  // OUT0204_I
          input  OUT3001_I : OUT_VOLTAGE_A_INPUT_MAPPING_TYPE  // OUT3001_I
          input  OUT3000_I : OUT_SUPPLY_A_INPUT_MAPPING_TYPE  // OUT3000_I
          input  OUT0001_I : OUT_PWM_25_B_INPUT_MAPPING_TYPE  // OUT0001_I
          input  OUT0003_I : OUT_PWM_25_B_INPUT_MAPPING_TYPE  // OUT0003_I
          input  OUT0005_I : OUT_PWM_25_B_INPUT_MAPPING_TYPE  // OUT0005_I
          input  OUT0101_I : OUT_PWM_25_B_INPUT_MAPPING_TYPE  // OUT0101_I
          input  OUT0103_I : OUT_PWM_25_B_INPUT_MAPPING_TYPE  // OUT0103_I
          input  OUT0105_I : OUT_PWM_25_B_INPUT_MAPPING_TYPE  // OUT0105_I
          input  OUT0201_I : OUT_PWM_25_B_INPUT_MAPPING_TYPE  // OUT0201_I
          input  OUT0203_I : OUT_PWM_25_B_INPUT_MAPPING_TYPE  // OUT0203_I
          input  OUT0205_I : OUT_PWM_25_B_INPUT_MAPPING_TYPE  // OUT0205_I
          input  OUT0007_I : OUT_PWM_40_BRIDGE_A_INPUT_MAPPING_TYPE  // OUT0007_I
          input  OUT0107_I : OUT_PWM_40_BRIDGE_A_INPUT_MAPPING_TYPE  // OUT0107_I
          input  OUT0207_I : OUT_PWM_40_BRIDGE_A_INPUT_MAPPING_TYPE  // OUT0207_I
          output OUT0006_Q : OUT_PWM_40_BRIDGE_A_OUTPUT_MAPPING_TYPE  // OUT0006_Q
          output OUT0106_Q : OUT_PWM_40_BRIDGE_A_OUTPUT_MAPPING_TYPE  // OUT0106_Q
          output OUT0206_Q : OUT_PWM_40_BRIDGE_A_OUTPUT_MAPPING_TYPE  // OUT0206_Q
          output OUT0008_Q : OUT_PWM_40_A_OUTPUT_MAPPING_TYPE  // OUT0008_Q
          output OUT0108_Q : OUT_PWM_40_A_OUTPUT_MAPPING_TYPE  // OUT0108_Q
          output OUT0208_Q : OUT_PWM_40_A_OUTPUT_MAPPING_TYPE  // OUT0208_Q
          output OUT0000_Q : OUT_PWM_25_A_OUTPUT_MAPPING_TYPE  // OUT0000_Q
          output OUT0002_Q : OUT_PWM_25_A_OUTPUT_MAPPING_TYPE  // OUT0002_Q
          output OUT0004_Q : OUT_PWM_25_A_OUTPUT_MAPPING_TYPE  // OUT0004_Q
          output OUT0100_Q : OUT_PWM_25_A_OUTPUT_MAPPING_TYPE  // OUT0100_Q
          output OUT0102_Q : OUT_PWM_25_A_OUTPUT_MAPPING_TYPE  // OUT0102_Q
          output OUT0104_Q : OUT_PWM_25_A_OUTPUT_MAPPING_TYPE  // OUT0104_Q
          output OUT0200_Q : OUT_PWM_25_A_OUTPUT_MAPPING_TYPE  // OUT0200_Q
          output OUT0202_Q : OUT_PWM_25_A_OUTPUT_MAPPING_TYPE  // OUT0202_Q
          output OUT0204_Q : OUT_PWM_25_A_OUTPUT_MAPPING_TYPE  // OUT0204_Q
          output OUT3001_Q : OUT_VOLTAGE_A_OUTPUT_MAPPING_TYPE  // OUT3001_Q
          output OUT3000_Q : OUT_SUPPLY_A_OUTPUT_MAPPING_TYPE  // OUT3000_Q
          output OUT0001_Q : OUT_PWM_25_B_OUTPUT_MAPPING_TYPE  // OUT0001_Q
          output OUT0003_Q : OUT_PWM_25_B_OUTPUT_MAPPING_TYPE  // OUT0003_Q
          output OUT0005_Q : OUT_PWM_25_B_OUTPUT_MAPPING_TYPE  // OUT0005_Q
          output OUT0101_Q : OUT_PWM_25_B_OUTPUT_MAPPING_TYPE  // OUT0101_Q
          output OUT0103_Q : OUT_PWM_25_B_OUTPUT_MAPPING_TYPE  // OUT0103_Q
          output OUT0105_Q : OUT_PWM_25_B_OUTPUT_MAPPING_TYPE  // OUT0105_Q
          output OUT0201_Q : OUT_PWM_25_B_OUTPUT_MAPPING_TYPE  // OUT0201_Q
          output OUT0203_Q : OUT_PWM_25_B_OUTPUT_MAPPING_TYPE  // OUT0203_Q
          output OUT0205_Q : OUT_PWM_25_B_OUTPUT_MAPPING_TYPE  // OUT0205_Q
          output OUT0007_Q : OUT_PWM_40_BRIDGE_A_OUTPUT_MAPPING_TYPE  // OUT0007_Q
          output OUT0107_Q : OUT_PWM_40_BRIDGE_A_OUTPUT_MAPPING_TYPE  // OUT0107_Q
          output OUT0207_Q : OUT_PWM_40_BRIDGE_A_OUTPUT_MAPPING_TYPE  // OUT0207_Q
      System_Inputs : System_Inputs, ifm electronic, version 3.0.0.1
          input  VBB30 : IN_SYSTEM_VOLTAGE_INPUT_MAPPING_TYPE  // VBB30
          input  VBB15 : IN_SYSTEM_VOLTAGE_INPUT_MAPPING_TYPE  // VBB15
          input  TemperatureBoard0 : IN_TEMPERATURE_INPUT_MAPPING_TYPE  // TemperatureBoard0
          input  TemperatureChip0 : IN_TEMPERATURE_INPUT_MAPPING_TYPE  // TemperatureChip0
      System_Outputs : System_Outputs, ifm electronic, version 3.0.0.1
          input  VBB0_SW_I : OUT_GROUP_SWITCH_INPUT_MAPPING_TYPE  // VBB0_SW_I
          input  VBB1_SW_I : OUT_GROUP_SWITCH_INPUT_MAPPING_TYPE  // VBB1_SW_I
          input  VBB2_SW_I : OUT_GROUP_SWITCH_INPUT_MAPPING_TYPE  // VBB2_SW_I
          output VBB0_SW_Q : OUT_GROUP_SWITCH_OUTPUT_MAPPING_TYPE  // VBB0_SW_Q
          output VBB1_SW_Q : OUT_GROUP_SWITCH_OUTPUT_MAPPING_TYPE  // VBB1_SW_Q
          output VBB2_SW_Q : OUT_GROUP_SWITCH_OUTPUT_MAPPING_TYPE  // VBB2_SW_Q
          output SUPPLY_SWITCH_Q : OUT_SYS_SWITCH_OUTPUT_MAPPING_TYPE  // SUPPLY_SWITCH_Q
  CR711S : CR711S, ifm electronic, order no. CR711S, version 3.0.0.1
  Project Information/
    function GetCompany [ST]
    function GetTitle [ST]
    function GetVersion [ST]
    function GetTextProperty [ST]
    function GetTextProperty2 [ST]
    function GetNumberProperty [ST]
    function GetBooleanProperty [ST]
    function GetVersionProperty [ST]
  text list GlobalTextList
*)

// StandardPLC/Application/DUTs/color
{attribute 'qualified_only'}
{attribute 'strict'}
{attribute 'to_string'}
TYPE color :
(
	red := 0,
	green := 1,
	blue := 2
);
(*(
	red,
	green,
	blue
);*)
END_TYPE

// StandardPLC/Application/POUs/GPS/eScrewParameters
//{attribute 'qualified_only'}
//{attribute 'strict'}
TYPE eScrewParameters :
(
	enum_member := 0,
	// Screw Parameters via pnezD field
	NS_PITCH := 1,
	SCREW_LENGTH := 2,
	TRUSS_VERT_ANGLE := 3, // tenth of deg; truss angle from vertical
	THIRD_LEG_VERT_ANGLE := 4, // tenth of deg, third leg angle from vertical - 8686 if no third leg
	EMBED_LENGTH := 5, // cm; length of embedment
	IE_MIN_HAMMER := 6, // cm; minimum hammering for intelligent embedment(IE)
	IE_MIN_EMBED := 7, // cm; min embedment for IE
	TRUSS_TYPE := 8, // Interior, Exterior, or Center: I,E,C
	
	// Truss types - correlate letters I,E,C to ascii numbers for direct conversion to real
	CENTER := 67,
	EXTERIOR := 69,
	INTERIOR := 73,
	
	NA := 222 // N/A this screw (eg if not a 3rd leg, 3rd leg angle from vertical would be 8686
);
END_TYPE

// StandardPLC/Application/DUTs/SqrStruct
TYPE SqrStruct :
STRUCT
	base: REAL := 7;
	//exponent: REAL := 2;
	pOut: POINTER TO REAL;
	
END_STRUCT
END_TYPE

// StandardPLC/Application/DUTs/Diag
{attribute 'qualified_only'}
// {attribute 'strict'} // why strict?
{attribute 'to_string'}
TYPE Diag :
(
	STAT_INACTIVE := 0, // POU is inactive. POU called with Enable / Execute = FALSE. 
	
	STAT_DONE := 1, // POU has finished processing successfully. Final results available and valid. 
	
	STAT_BUSY := 2, // POU is still processing. Final result not yet available.
	
	// However, some outputs may be updated each cycle.
	 
	
	STAT_PREPARING := 3, // POU is still proccessing. Final result not yet available.
	
	(*However, some outputs may be updated each cycle.
	
	This value is used in ‘Enable’ behaviors instead of the STAT_BUSY status,
	
	to be distinct from ‘Execute’ behaviors.*)
	 
	
	STAT_READY := 4, // POU is initialised and ready to execute other commands.
	
	STAT_RESET := 5, // POU is processing reset operations.
	
	STAT_ABORTED := 6, // Reserved for later usage 
	
	RESERVED_07 := 7, // Reserved for later usage 
	
	RESERVED_08 := 8, // Reserved for later usage 
	
	RESERVED_09 := 9, // Reserved for later usage 
	
	ERR_OPEN_CIRCUIT := 10, // Open circuit detected. Possible wire break. 
	
	ERR_SHORT_CIRCUIT := 11, // Short circuit TO GND OR VBBx detected. 
	
	ERR_OVERLOAD_CURRENT := 12, // Current above allowed maximum detected. 
	
	ERR_LOW_CURRENT := 13, // Current below allowed minimum detected. 
	
	ERR_UNDERVOLTAGE_VBBX := 14, // For inputs: Critical under voltage at reference.
	
	// For outputs: Critical under voltage at responsible OutputGroup supply or at VBB30 / VBB15.
	 
	ERR_OVERVOLTAGE_VBBX := 15, // For inputs: Critical over voltage at reference.
	
	// For outputs: Critical over voltage at responsible OutputGroup supply or at VBB30 / VBB15.
	 
	ERR_STUCK_AT_HIGH := 16, // Stuck-at-high detected. 
	
	ERR_STUCK_AT_LOW := 17, // Stuck-at-low detected. 
	
	ERR_HIGH_TEMPERATURE := 18, // Board temperature exceeded maximum threshold. 
	
	ERR_LOW_TEMPERATURE := 19, // Board temperature undercut minimum threshold. 
	
	ERR_INVALID_VALUE := 20, // One or more input parameters are invalid or exceeding their allowed range. 
	
	ERR_INVALID_CHANNEL := 21, // Channel not available. 
	
	ERR_INVALID_MODE := 22, // Mode not available or not supported by this channel. 
	
	ERR_INVALID_FREQUENCY := 23, // Frequency not supported for active mode. 
	
	ERR_INVALID_DITHER := 24, // One or more dither parameters are invalid. 
	
	ERR_INVALID_FILTER := 25, // One or more filter parameters are invalid. 
	
	ERR_UNREACHABLE_CURRENT := 26, // Current control can not reach desired current. 
	
	ERR_SLOW_SIGNAL := 27, // Input signal is too slow for measurement. 
	
	ERR_CHANGEOVER_TIME := 28, // Changeover time for driver protection not yet expired. 
	
	ERR_INSTANCE := 29, // The passed instance was NULL or invalid. (e.g. FB object was NULL.) 
	
	ERR_INSTANCE_LIMIT := 30, // Instance limit reached. 
	
	ERR_INVALID_COLOUR := 31, // Value for colour of LED is not valid. 
	
	ERR_NO_IDENTITY := 32, // Application/User identity is currently not set. 
	
	ERR_ACCESS := 33, // The requested resource could not be registered for write access for the calling PLC,
	
	// because it is already registered for write access by another PLC.
	
	ERR_UNDEFINED := 34, // The called function returned a result value that is not mapped to any end-user result.  Please inform your supplier.
	 
	
	ERR_FUNC_KEY_MISSED := 35, // TODO 
	
	ERR_BUFFER_OVERFLOW := 36, // Tx or Rx buffer overflow. Message could not be written to Tx buffer
	
	// or one or more messages could not be written to Rx buffer and were lost.
	 
	
	ERR_BAUDRATE_ALREADY_SET := 37, // The desired baud rate could not be set, because there is already another baud rate defined. 
	
	ERR_INACTIVE_INTERFACE := 38, // Chosen interface is not enabled or not intialized. 
	
	ERR_TIMEOUT := 39, // The allowed maximum execution time has been exceeded. Action could not complete. 
	
	ERR_OUT_OF_MEMORY := 40, // TODO 
	
	ERR_BUS_OFF := 41, // CAN interface is in the state ‘bus off’. 
	
	ERR_BAD_CRC := 42, // CRC of an accessed memory area is invalid. Read data is invalid. 
	
	ERR_EXCEEDED_RANGE := 43, // An output value exceeds the displayable range of its data type.
	
	// Displayed value will be limited to the data types respective MIN or MAX value.
	 
	
	ERR_INTERNAL_COMMUNICATION := 44, // An internal called low level function reports an error (e.g. low level library version mismatch) 
	
	ERR_NOT_SUPPORTED := 45, // Invalid call. Function is not supported by the runtime. 
	
	ERR_TIMING := 46, // Signal endges in an unexpected order detected. 
	
	ERR_INTERNAL := 47, // Internal system error. 
	
	ERR_FILE_SYSTEM := 48, // File operation has failed. 
	
	ERR_INVALID_IP_CFG := 49, // Invalid IP address or Netmask or gateway configured 
	
	ERR_FAILED_ERR_RESET := 50, // OBSOLETE. Kept for backwards compatibility. 
	
	ERR_DEVICE_NOT_AVAILABLE := 51, // Selected Device e.b. USB device is not available 
	
	ERR_NO_OBJECT := 52, // No object with this specified name available. Ex: file name specified not available to open or get size 
	
	ERR_UNREACHABLE_VOLTAGE := 53, // Voltage control cannot reach desired voltage 
	
	ERR_AT_GROUP_OUTPUT := 54, // One or more outputs of the output group are in error state 
	
	ERR_CONTROL_DITHER := 55, // The requested dither value could not adjusted 
	
	ERR_UNDERVOLTAGE_VBBX_WARNING := 56, // OBSOLETE. Kept for backwards compatibility. Use DIAG_UNDERVOLTGE_VBBX instead. 
	
	ERR_OVERVOLTAGE_VBBX_WARNING := 57, // OBSOLETE. Kept for backwards compatibility. Use DIAG_OVERRVOLTGE_VBBX instead. 
	
	ERR_LOW_TEMPERATURE_WARNING := 58, // OBSOLETE. Kept for backwards compatibility. Use DIAG_LOW_TEMPERATURE instead. 
	
	ERR_HIGH_TEMPERATURE_WARNING := 59, // OBSOLETE. Kept for backwards compatibility. Use DIAG_HIGH_TEMPERATURE instead. 
	
	ERR_RANGE_OVERRUN := 60, // Measured Value (input / output, current / voltage) exceeds set higher limit given by application. 
	
	ERR_RANGE_UNDERRUN := 61, // Measured Value (input / output, current / voltage) undercuts set lower limit given by application. 
	
	DIAG_INVALID_VALUE := 62, // One or more input parameters are invalid or exceeding their allowed range. 
	
	DIAG_INTERNAL := 63, // OBSOLETE. Kept for backwards compatibility. Use ERR_INTERNAL instead. 
	
	DIAG_OPEN_CIRCUIT := 64, // Open circuit detected. Possible wire break. (if protection disabled) 
	
	DIAG_SHORT_CIRCUIT := 65, // Short circuit to GND or VBBx detected. (if protection disabled) 
	
	DIAG_UNDERVOLTAGE_VBBX := 66, (*For inputs: Critical under voltage at reference (if protection disabled).
	
	For outputs: Critical under voltage at responsible OutputGroup supply or at VBB30 / VBB15.
	
	(if protection disabled) *)
	 
	
	DIAG_OVERVOLTAGE_VBBX := 67, (* For inputs: Critical over voltage at reference (if protection disabled).
	
	For outputs: Critical over voltage at responsible OutputGroup supply or at VBB30 / VBB15.
	
	(IF protection disabled)*)
	 
	
	DIAG_OVERLOAD_CURRENT := 68, // Current above allowed maximum detected. (if protection disabled) 
	
	DIAG_STUCK_AT := 69, // Stuck-at deteceted with no distinctive direction. (if protection disabled) 
	
	DIAG_STUCK_AT_HIGH := 70, // Stuck-at-high detected. (if protection disabled) 
	
	DIAG_STUCK_AT_LOW := 71, // Stuck-at-low detected. (if protection disabled) 
	
	DIAG_INVALID_COLOUR := 72, // Value for colour of LED is not valid. 
	
	DIAG_OVERVOLTAGE := 73, // Measured input- or output voltage exceeded maximum limit. (if protection disabled) 
	
	DIAG_UNDERVOLTAGE := 74, // Measured input- or output voltage undercut minimum limit. (if protection disabled) 
	
	DIAG_NO_CALIB := 75, // IO has no valid calibration. Default values used. 
	
	DIAG_ACCESS := 76, // Addressed resource is not owned by calling PLC. 
	
	DIAG_CHANGEOVER_TIME := 77, // Minimum changeover time for highside <–> lowside switching of drivers not yet expired. 
	
	ERR_OVERVOLTAGE := 78, // Measured input- or output voltage exceeded maximum limit. 
	
	ERR_UNDERVOLTAGE := 79, // Measured input- or output voltage undercut minimum limit. 
	
	ERR_STUCK_AT := 80, // Stuck-at deteceted with no distinctive direction. 
	
	DIAG_CONTROL_DITHER := 81, (* The requested dither value could not be adjusted because the result of dither
	
	and the given PWM value is higher than 1000 per mill.*)
	 
	
	DIAG_SLOW_SIGNAL := 82, // Input signal is too slow for measurement. 
	
	DIAG_DIAG_PRO_MODE := 83, // Invalid or unsupported diagnosis-protection mode. 
	
	DIAG_WINDOW := 84, // Invalid values for user diagnosis window. 
	
	ERR_SDO_IDX_NOT_EXIST := 85, // SDO index does not exist. 
	
	ERR_SDO_SUBIDX_NOT_EXIST := 86, // SDO sub-index ndoes not exist. 
	
	ERR_SDO_UNSUPPORTED_ACCESS := 87, // SDO access is not supported. 
	
	ERR_SDO_DATA_TYPE := 88, // Wrong SDO data type. 
	
	DIAG_LOW_TEMPERATURE := 89, // Board temperature undercut minimum warning threshold. 
	
	DIAG_HIGH_TEMPERATURE := 90, // Board temperature exceeded maximum warning threshold. 
	
	DIAG_INVALID_DITHER := 91, // One or more dither parameters are invalid. 
	
	DIAG_INVALID_FREQUENCY := 92, // Frequency not supported for active mode. 
	
	DIAG_RANGE_OVERRUN := 93, // Measured Value (input / output, current / voltage) exceeds set higher limit given by application 
	
	DIAG_RANGE_UNDERRUN := 94, // Measured Value (input / output, current / voltage) undercuts set lower limit given by application. 
	
	DIAG_INVALID_FILTER := 95, // One or more filter parameters are invalid. 
	
	ERR_COMPARE_MISMATCH := 96, (* Mismatch detected between the mission- and monitor values of the selected resource.
	
	Example: A 2-channel function like safe input or OSSD input has read an actual value that is outside
	
	of the specified tolerance band of the expected value.*)
	 
	
	DIAG_INVALID_IP_CFG := 97, // Invalid IP address or netmask or gateway configured. 
	
	DIAG_LOW_CURRENT := 98, // Current below allowed minimum warning level detected. 
	
	DIAG_AT_GROUP_OUTPUT := 99, // One or more outputs of the output group are in error state. (when protection disabled) 
	
	ERR_SDO_UNKNOWN := 100, // SDO access NOT successful. Reason unknown 
	
	ERR_BAUDRATE_INVALID_OR_ALREADY_SET := 101, // The desired baud rate could not be set because it’s invalid or there is already another baud rate defined at the selected channel. 
	
	DIAG_COMPARE_MISMATCH := 102, // Mismatch detected between the mission- and monitor values of the selected resource. 
	
	DIAG_COMPARE_MISMATCH_VSYS := 103, // Mismatch detected between the mission- and monitor values of the selected system voltage resource. 
	
	DIAG_GROUP_OVERLOAD_CURRENT := 104, // Current at output group above allowed maximum detected. 
	
	ERR_GROUP_OVERLOAD_CURRENT := 105, // Current at output group above allowed maximum detected. 
	
	STAT_PAUSED := 106, //: One or more operations is paused. Example: media playing or media recording 
	
	STAT_ABORT := 107, //: FB is executing ABORT sequence before completing the defined task, the end results are unpredictable 
	
	STAT_EVNT_OPEN_PLUG_STORAGE := 108, //: FB is opening call back event for mounting event of storage devices 
	
	STAT_EVNT_OPEN_UNPLUG_STORAGE := 109, //: FB is opening call back event for removal event of mounted storage devices 
	
	STAT_EVNT_OPEN_DONE := 110, //: Call back event opening is done 
	
	STAT_EVNT_REGI_PLUG_STORAGE := 111, //: FB is registering a call back function for mounting event of storage devices 
	
	STAT_EVNT_REGI_UNPLUG_STORAGE := 112, //: FB is registering a call back function for removal event of mounted storage devices 
	
	STAT_EVNT_REGI_DONE := 113, //: Call back function registration is done 
	
	STAT_EVNT_UNREGI := 114, //: FB is unregistering the call back function 
	
	STAT_EVNT_UNREGI_DONE := 115, //: Call back function unregistering is done 
	
	STAT_EVNT_CLOSE := 116, //: FB is closing the call back event 
	
	STAT_EVNT_CLOSE_DONE := 117, //: Call back event closing is done 
	
	ERR_INSTANCE_RESTRICTION := 118, //: This FB is restricted to use along with some other FB, Read the FB description for more details 
	
	ERR_NO_FILE := 119, //: No file with this specified name available 
	
	ERR_EVNT_OPEN := 120, //: Error while opening an event for call back function registration 
	
	ERR_EVNT_REGI := 121, //: Error while registering a call back function for a call back event 
	
	ERR_EVNT_UNREGI := 122, //: Error while unregistering a call back function for a call back event 
	
	ERR_EVNT_CLOSE := 123, //: Error while closing an event that was was opened for call back function registration 
	
	ERR_GET_STORAGE_LIST := 124, //: Error while reading list of mounted storage devices 
	
	ERR_UNPLUG_STORAGE := 125, //: Error while removing a mounted storage devices 
	
	DIAG_INVALID_CHANNEL := 126, //: Channel not available. 
	
	DIAG_INVALID_MODE := 127, //: Mode not available or not supported by this channel. 
	
	ERR_H_BRIDGE_TEST := 128, //: H-Bridge test failed. 
	
	ERR_GROUP_SW_TEST := 129, //: Group swirch test failed. 
	
	ERR_TX_ERROR := 130, //: Sending message faild. 
	
	ERR_RX_ERROR := 131 //: Receiving message failed. Data was lost. 
	
);

END_TYPE

// StandardPLC/Application/POUs/Utilities/ProfileGen/CurveTypes
{attribute 'qualified_only'}
{attribute 'strict'}
TYPE CurveTypes :

(
	// var := independent variable
	// x := characteristic value
	LINEAR := 1, // x*var
	INVERSE := 2, // x/var
	EXPONENT := 3, // var^x
	EXPONENTIAL := 4, // x^var
	LOGB10 := 5, // x*LOG(var)
	NATLOG := 6, // x*ln(var)
	SIGMOID := 7, // [(var-x)/(sqrt(1+(var-x)2] + 1 until the midpoint, then [((1-var)-x)/(sqrt(1+((1-var)-x)2] + 1;
	RES1 := 8,
	RES2 := 9,
	RES3 := 10
);

END_TYPE

// StandardPLC/Application/POUs/Utilities/ProfileGen/TDcontrolCode/sSetpoint
TYPE sSetpoint :
STRUCT
	(* User side setpoints are in engineering units *)
	POSITION_ENGR: REAL;
	VELOCITY_ENGR: REAL;
	ACCELERATION_ENGR: REAL;
	(* Internal use setpoint are in counts *)
	POSITION_RAW: DINT;
	VELOCITY_RAW: REAL;
	ACCELERATION_RAW: REAL;
	(* Flag to allow the profiler know a new setpoint is in *)
	SETPOINT_CHANGED: BOOL;
END_STRUCT
END_TYPE

// StandardPLC/Application/POUs/Utilities/ProfileGen/TDcontrolCode/sFeedback
TYPE sFeedback :
STRUCT
	(* Whether or not this axis has an installed feedback device. *)
	INSTALLED: BOOL := FALSE;
	(* Raw feedback counts per engineering unit *)
	RAW_PER_ENGR: REAL := 1.0;
	(* Encoder counts when engineering units are zero *)
	RAW_WHEN_ENGR_ZERO: DINT := 0;
	(* Maximum valid feedback, raw counts.  Set min and max to 0 to disable! *)
	FEEDBACK_VALID_MAX: DINT := 0;
	(* Minimum valid feedback, raw counts.  Set min and max to 0 to disable! *)
	FEEDBACK_VALID_MIN: DINT := 0;

	POSITION_RAW: DINT := 0;
	POSITION_ENGR: REAL := 0.0;
	VELOCITY_RAW: REAL := 0.0;
	VELOCITY_ENGR: REAL := 0.0;
	US_LAST_SAMPLE: DWORD := 0;
	POSITION_RAW_LAST_SAMPLE: DINT := 0;
	VALID: BOOL := FALSE;
	SAMPLE_VALID: BOOL := FALSE;
	COUNT: UDINT := 0;
	ROLLOVER_AT: DINT := 0;
	ROLLOVER_HALF: DINT := 0;
	
	ABS_ZERO_ABOVE_RANGE_HALF: BOOL := FALSE;
	ABS_RANGE_MIN: DINT := 0;
	ABS_RANGE_MAX: DINT := 0;

	//VELOCITY_CALC_01: VELOCITY_CALC;
END_STRUCT
END_TYPE

// StandardPLC/Application/POUs/GPS/eGPS

TYPE eGPS : // 0 - 15 positions with GPS_AUTOTARGET_STATUS as UINT
(
	GPS_WP_AUTOTARGET_ON := 0,
	GPS_HEADING := 1,
	GPS_X := 2,
	GPS_Y := 3,
	GPS_Z := 4,
	GPS_AXIS_NOT_IN_RANGE := 5,
	GPS_AXIS_NOT_IN_RANGE_NOT_IN_AUTO := 6,
	GPS_AXIS_IN_RANGE := 7,
	GPS_AXIS_ON_TARGET := 8,
	GPS_AXIS_SETTLED_WITHIN_TARGET_BAND := 9,
	ALL_GPS_AXES_IN_RANGE := 10,
	ALL_GPS_AXES_ON_TARGET := 11,
	GPS_STABLE_5S := 12, // Gps fixed solution over 5s with 5 checks per second
	GPS_USED_THIS_TRUSS := 13 // decision per truss whether gps autotargeting being used
	
	
);

END_TYPE

// StandardPLC/Application/POUs/GPS/eGpsDataCategories
{attribute 'qualified_only'}
{attribute 'strict'}
TYPE eGpsDataCategories :
(
	GPS_AXIS_AUTOTARGET_ON := 0,
	GPS_AXIS_RANGE := 1,
	GPS_AXIS_TARGET := 2
);
END_TYPE

// StandardPLC/Application/DUTs/Coordinates2d
TYPE Coordinates2d :
STRUCT
	x: REAL;
	y: REAL;
END_STRUCT
END_TYPE

// StandardPLC/Application/DUTs/Coordinates3d
TYPE Coordinates3d :
STRUCT
	x: REAL;
	y: REAL;
	z: REAL;
END_STRUCT
END_TYPE

// StandardPLC/Application/POUs/GPS/sGPSaxis
TYPE sGPSaxis : // changes made here must also be made in HMI code
STRUCT
	
	OFFSET: REAL := 0;                      // distance to move to target as indicated by GPS
	SMOOTHED_OFFSET: REAL := 0;		        // averaged over a short time (eg 0.1s, or 5 cycles)
	OFFSET_WORLD_FRAME: REAL := 0;          // off set in reference to wp as origin in world frame vs TD frame
	OFFSET_WORLD_FRAME_FILTERED: REAL := 0; // off set in reference to wp as origin in world frame vs TD frame
	REACH: REAL := 0;                       // furthest distance at which actuator will use gps to autotarget
	TARGET_LIMIT: REAL := 0;                // furthest distance at which axis is considered to be satisfactorily on target
	AUTOTARGET_ON: BOOL := FALSE;           // whether autotarget is activated for this axis
	 
	 (* Range status:
		0: not in range to auto-target; 
		1: in range to move to target but not on target, OR autotarget not selected;
		2: in range to move to target, not on target; 
		3: within target specification; 
		4: settled withinFixedBand of target specification (settled over designated time);
		*)
	RANGE_STATUS: UINT := 0;   
    SETTLED_WITHIN_BAND: BOOL := FALSE;  
	VEL: REAL :=0;
	ACCEL: REAL := 0;
	TARGET_POSITION: REAL := 0;
	AXIS_RANGE_MAX: REAL := 0;
	AXIS_RANGE_MIN: REAL := 0;
END_STRUCT
END_TYPE

// StandardPLC/Application/DUTs/sScrewParams
TYPE sScrewParams :
STRUCT
(*
	This structure is used to store pnezD descriptions as well as custom recipes if changes need to be made in the field
*)
NS_PITCH : SINT := 0;
SCREW_LENGTH : UINT := 0;
TRUSS_VERT_ANGLE : USINT := 0;
THIRD_LEG_VERT_ANGLE : USINT := 0;
EMBED_LENGTH : USINT := 86;
IE_MIN_HAMMER : USINT := 86;
IE_MIN_EMBED : USINT := 86;
TRUSS_TYPE : USINT := 0;

END_STRUCT
END_TYPE

// SafetyPLC/Application/EVL
(* THIS EVL IS AUTOGENERATED. DO NOT MODIFY THESE ATTRIBUTES. *)
{attribute 'location' := '16#800' }
{attribute 'linkalways'}
{attribute 'qualified_only'}
VAR_GLOBAL

END_VAR

// StandardPLC/Application/GlobalVars/Test1Vars
//{attribute 'qualified_only'}
VAR_GLOBAL

	//: ARRAY [0..100] OF UINT := [100(0)];
	debug: ARRAY [0..100] OF REAL := [100(0)];
	debug_word: ARRAY [0..100] OF WORD := [100(0)];
	
	// ddtLayers test
	Target_result: REAL := 0;
	Start_test: BOOL := FALSE;
END_VAR

// StandardPLC/Application/Network Variables/PLC_TRANSMIT_1
{attribute 'qualified_only'}
VAR_GLOBAL
	
END_VAR

// StandardPLC/Application/GlobalVars/Test2Vars
//{attribute 'qualified_only'}
VAR_GLOBAL
		
	test1 : INT;
	test2 : INT;
	test3 : INT;
	test4 : INT;

		WIRED_OUTS: ARRAY [1..4] OF POINTER TO INT :=
	[
		ADR(test1),       //1
		ADR(test2),       //2
		ADR(test3),       //3
		ADR(test4)        //4

	];
	
END_VAR

// StandardPLC/Application/GlobalVars/Dims
//{attribute 'qualified_only'}
VAR_GLOBAL
	// generic
	Pi : REAL := 3.14159265;
	
	// TD2
	
	// TD3
	YAW_ARM_LENGTH: REAL := 135;
	BS_LENGTH: REAL := 135;
	BS_PIVOT_TO_YAW_PIVOT: REAL := 135; // aka BS_LENGTH
	YAW_PIVOT_TO_DRILL_ROD: REAL := 135;
	
END_VAR

// StandardPLC/Application/GlobalVars/Positions
//{attribute 'qualified_only'}
VAR_GLOBAL // all perspectives from operator position facing target plate at rear of truss driver
	
	// TD3 positions
	BOOM_SWING_ANGLE: REAL := 0; // + deg to RIGHT, - to LEFT; +/- 24 deg
	X_SLIDE_POS: REAL := 15; // 0 forward to 30 cm rear toward operator
	YAW_ANGLE: REAL := 0; // + deg to LEFT, - to RIGHT, opposite of BS; +/- 24 deg
	Z_SLIDE_POS: REAL := 105; // 2 to 167.5 cm low to high
	
	(* 	target offsets per gps in reference to TD wp
		x + means move forward; y means move right; z + means move up; 
		Heading + means ccw from pivot, or move operator end right
	*)
	// GPS positions
	// [ Heading, X, Y, Z, spare, spare ]
	GPS_AXES: ARRAY [1..6] OF sGPSaxis; // set to greater than NUM_GPS_AXES; 
	NUMBER_GPS_AXES: INT := 4; // set = to NUM_GPS_AXES
	
	(* Imaginary world coordinate system: ( correlates to TD aligned N - S with operator end on North side )
			Heading  (H): + is CCW from North
			Northing (X): + is North
			Easting  (Y): + is East
			Altitide (Z): + is up
		default is TD at (H,N,E,Z): (0,0,0,0)
	*)
	GPS_HEADING_OFFSET: REAL := 77.7;
	GPS_X_OFFSET: REAL := 77.7;
	GPS_Y_OFFSET: REAL := 77.7;
	GPS_Z_OFFSET: REAL := 77.7;
	HEADING_TO_TARGET_OFFSET: REAL := 0;
	
	
END_VAR

// StandardPLC/Application/GlobalVars/GPS_Data
//{attribute 'qualified_only'}
VAR_GLOBAL
	// GPS
	GPS_VENDOR: UINT := 0;
	
	(*                  --  GPS AUTO TARGET BOOLS:  --
		GPS_AUTOTARGET_STATUS.0 = WP AUTO-TARGET bool - no axis will autotarget without this set
							 .1 - .9 = select axes Auto target bools: .1 = heading, .2 = x, .3 = y, .4 = z
							 .10: all gps axes are in range for autotarget
							 .11: all gps axes are on target  
							 .12: gps fixed solution for 5s and autotarget on                                                              *)
	GPS_AUTOTARGET_SELECTION: UINT := 0; 
	
	(*:= [Heading in range,    	       Heading on target        
		  X "",                		   X ""
		  Y "",          			   Y ""
		  Z "",           			   Z ""
		  velocity factor,  		   accel factor, 
		  radio delay warning,		   radio delay critical, 
		  Number of retargets,         reserved]   
	      7,8 correlate to eGPS enum labels *)
	GPS_SETTINGS: ARRAY [1..12, 7..8] OF REAL := [15, 0.30, 8, 9, 15, 12, 82, 12, 0.9, 0.5, 3, 5, 0.7, 3, 10(8888)];
	GPS_SIM_OFFSETS: ARRAY [1..4] OF REAL := [0, 0, 0, 0]; // offsets in mm
	
	// [ All, Heading, x, y, z ]
	GPS_IN_RANGE: ARRAY [0..4] OF BOOL := [5(0)];
	TARGET_POSITIONS_METHOD_1: ARRAY [1..4] OF REAL := [4(0)];
	TARGET_POSITIONS_METHOD_2: ARRAY [1..4] OF REAL := [4(0)];
	
	// temp debug
	GPS_RANGE_MARGIN: REAL;
	PERCENT_MARGIN_AS_FACTOR: REAL;
	ROTATE_DEG_FROM_YAW_TO_BS: REAL := 0; // How many degrees to rotate coordinate system to align with boom swing
	
	// temp debug GpsTdToWorldFixAll2d
	BS_ANGLE_NS_DELTA: REAL := 0;
	BS_ANGLE_WORLD_NS: REAL := 0;
	BS_ANGLE_NS_TO_Y_TARGET_DELTA: REAL := 0;
	
	X_OFFSET: REAL := 0; // offsets from WP given by gps, in TD frame, + is forward of operator 
	Y_OFFSET: REAL := 0; // + is to the right of operator (facing forward at rear [mast end] of TD)
	YAW_OFFSET: REAL := 0; // heading offset to rotate by as given by gps, + is moving mast to the right (CCW) of operator
	X_OFFSETS: ARRAY [1..9] OF REAL := [9(0)];
	Y_OFFSETS: ARRAY [1..9] OF REAL := [9(0)];
	YAW_OFFSETS: ARRAY [1..9] OF REAL := [9(0)];
	
	HEADING_TO_TARGET: REAL := 0;
	
	//GPS AutoTrack
	GPS_LEFT_JS: INT := 0;	
	GPS_RIGHT_JS: INT := 0;
	GPS_LEFT_POSITIVE: BOOL := TRUE;	
	GPS_RIGHT_POSITIVE: BOOL := TRUE;	
	
	// PNEZD
	GPS_PNEZD_P: STRING(16); // "Pole id"
	GPS_PNEZD_N: REAL := 0; // Northing
	GPS_PNEZD_E: REAL := 0; // Easting
	GPS_PNEZD_Z: REAL := 0; // "Vertical"
	GPS_PNEZD_D: STRING(64); // "Description"
	
	// debug
	LEFT_TRACK_OUTPUT: REAL := 0;
	RIGHT_TRACK_OUTPUT: REAL := 0;
	
	GPS_READY: BOOL := TRUE;
	
	//parameters from pnezD D field
	SCREW_PARAMETERS: ARRAY [1.. NUM_SCREW_PARAMETERS] OF REAL := [NUM_SCREW_PARAMETERS(6666)];
	SCREW_PARAMS_CUSTOM: ARRAY [0.. NUM_SCREW_PARAMETERS] OF sScrewParams;

	
	(*Screw lengths and count: [screw lengths, screw count] 
	 this list will self populate new screws until the max of SCREW_LENGTHS_COUNT is reached *)
	SCREW_COUNT: ARRAY [1..2, 1..SCREW_LENGTHS_COUNT] OF UDINT := [SCREW_LENGTHS_COUNT(0),SCREW_LENGTHS_COUNT(0)];
	
END_VAR

// StandardPLC/Application/GlobalVars/Ojjo_TD

VAR_GLOBAL CONSTANT
	// 20 millisecond cycle task executes all machine control functions.
	CONTROL_FREQ_HZ: REAL := 50.0;
	// This is hardcoded in the HMI code as constants can't be transmitted.
	UR_STALL_WINDOW_MAX: REAL := 2.0;
	SS_DETECT_WINDOW_MAX: REAL := 5.0;
	FLOW_TABLE_SIZE: INT := 5;

	(* ------------------------ No handling in language unfortunately ----------------------------------------*)
	SMALLEST_REAL: REAL := -3.402823E+38;
	LARGEST_REAL: REAL := 3.402823E+38;
	NUM_GPS_AXES: INT := 4; 
	NUM_SCREW_PARAMETERS: INT := 8; // number of screw parameters coded by pnezD field
	SCREW_LENGTHS_COUNT: USINT := 18;
END_VAR

VAR_GLOBAL
	(* ------------------------ TIME TRACKING ----------------------------------------*)
	TIME_SECONDS: DWORD;
	MSTIME: DWORD;
	CYCLE_TIME_START: REAL := 0.0;
	CYCLE_START: DWORD := 0;

	(* ----------------------- DEBUGGING CONTROL ------------------------------------ *)
	SIMULATION: BOOL := FALSE;
	SIMULATED_TIME_US: DWORD := 12345678;
	DEBUG_LC_STALL_DETECTED: BOOL := FALSE;
	DEBUG_UR_STALL_DETECTED: BOOL := FALSE;
	DEBUG_HARD_SOIL_DETECTED: BOOL := FALSE;

	(* ---------------------- GLOBAL HARDWARE AND CONTROL ------------------------------ *)
	(*
	pNVM1: POINTER TO sPersistent_1 := ADR(%MB0);
	pNVM2: POINTER TO sPersistent_2;
	pNVM3: POINTER TO sPersistent_3;
	pNVM4: POINTER TO sPersistent_4;
	*)
	
	AUTOMATIC_ALLOWED: BOOL := TRUE;
	FEEDBACK_FAILED: BOOL := FALSE;
	ANY_VALVE_FAILED: BOOL := FALSE;
	BV: REAL;
	
	BASE_ROLL_FILTERED_SLOW: REAL;
	BASE_PITCH_FILTERED_SLOW: REAL;
	BASE_ROLL_FILTERED_FAST: REAL;
	BASE_PITCH_FILTERED_FAST: REAL;
	
	HORN_REQUEST_TIMES: INT;
	HORN_REQUEST_OFF: TIME;
	HORN_REQUEST_ON: TIME;
	HORN_REQUEST_LAST_STATE: BOOL;
	
	MACHINE_STATE_STRING: STRING;
	METHOD_STRING: STRING;
	ERROR_STRING_SHORT: STRING;
	WARNING_STRING_SHORT: STRING;
	
	// Address to be used where necessary.
	J1939_ADDRESS: USINT := 47;
	
	(* ---------------------- TRACK MODE STATES and DATA HERE ---------------------- *)
	TRACK_STATE: eTrackStates;
	TRACK_MODE_STATE_CHANGE: BOOL := FALSE;

	TRACK_LEFT_TIME: INT := 0;
	TRACK_RIGHT_TIME: INT := 0;
	TRACK_BACK_TIME: INT := 4000;

	TRACK_BACK_REQUIRED: BOOL := FALSE;

	(* ---------------------- SCREW MODE STATES and DATA HERE ---------------------- *)
	SCREW_STATE: eScrewStates;
	SCREW_MODE_STATE_CHANGE: BOOL := FALSE;
	SCREW_MODE_PAUSED: BOOL := FALSE;
	SCREW_MODE_PAUSED_CHANGE: BOOL := FALSE;
	SCREW_DRIVE_DONE: BOOL := FALSE;
	SCREW_EMBEDDED_VISUAL: BOOL := FALSE;
	SCREW_START_POS: REAL;

	COMPRESSOR_REQUEST: BOOL := FALSE;

	UPPER_CROWD_REVEALING: BOOL := FALSE;
	UPPER_CROWD_DONE_REVEALING: BOOL := FALSE;
	BRIEF_HAMMER_START: REAL;

	(* Latched values for screw driving operation. *)
	WP_HEIGHT_LATCH: eWorkpointHeight;
	SCREW_LENGTH_LATCH: eScrewLength;
	SCREW_LENGTH_CM: REAL := 150.0;

	(* Latched position values when entering screw mode. *)
	MAST_SLIDE_AT_WP: REAL;
	LOWER_CROWD_AT_WP: REAL;

	(* Screw drive calculation variables. *)
	SCREW_REF_FROM_WP_EMBED: REAL := 0.0;

	CROWD_EMBED_ENDPOINT: REAL := 0.0;
	CROWD_ADVANCE_MIN: REAL := 0.0;
	SCREW_EMBEDMENT: REAL := 0.0;

	LEG_LENGTH_EMBED: REAL := 0.0;
	LEG_LENGTH_ACTUAL: REAL := 0.0;
	LEG_OVERDRIVE: REAL := 0.0;

	ROTATOR_CENTER_TO_GROUND: REAL;
	DRILL_TIP_BELOW_ROTATOR: REAL;
	
	(* Screw driving data. *)
	LOWER_CROWD_VEL_SMOOTHED: REAL := 0.0;		(* Lower rotary uses a smoothed version of the lower crowd velocity to remove some noise when following. *)
	LOWER_CROWD_POS_RAW: UDINT := 0;
	LOWER_CROWD_VEL_RAW: INT := 0;
	
	(* ------ All the fucked up stuff for workpoints that can't be reached by the rotator is here. ------ *)
	BOOM_SWING_AT_WP: REAL;
	YAW_AT_WP: REAL;
	Z_SLIDE_AT_WP: REAL;
	X_SLIDE_AT_WP: REAL;
	
	(* NXT 3 legged motor truss values here. *)
	BOOM_SWING_DELTA: REAL := 0.0;
	NXT_3LM_X_SLIDE_LEFT: REAL;
	NXT_3LM_X_SLIDE_RIGHT: REAL;
	NXT_3LM_Z_SLIDE_LEFT: REAL;
	NXT_3LM_Z_SLIDE_RIGHT: REAL;
	NXT_3LM_BOOM_SWING_LEFT: REAL;
	NXT_3LM_BOOM_SWING_RIGHT: REAL;
	NXT_3LM_YAW_LEFT: REAL;
	NXT_3LM_YAW_RIGHT: REAL;
	
	(* These are Y and Z relative to the BR pivot. *)
	WP_Y: REAL;
	WP_Z: REAL;
	ROTATOR_WP_Y: REAL;
	ROTATOR_WP_Z: REAL;
	ROTATOR_Y: REAL;
	ROTATOR_OFFSET_Y: REAL;
	BOOM_SWING_SCREW: REAL;
	Z_SLIDE_SCREW: REAL;
	LOW_WP_ADJUST: REAL;

	(* ----------------------- SCREW MODE: Machine pitch ------------------------------ *)
	BASE_PITCH_START: REAL := 0.0;
	BASE_PITCH_END: REAL := 0.0;
	KNUCKLE_PITCH_START: REAL := 0.0;
	KNUCKLE_PITCH_END: REAL := 0.0;
	MANDREL_PITCH_ERROR: REAL := 0.0;

	(* ----------------------- SCREW MODE: Compliance preload ------------------------------ *)
	PRELOAD_COMPLETE: BOOL := FALSE;
	PRELOAD_ANGLE_START: REAL := 0.0;
	PRELOAD_DELTA_CURRENT: REAL := 0.0;
	PRELOAD_MOTION_MAX: REAL := 30.0; // Maximum mast slide motion to preload.
	PRELOAD_MOTION_LIMIT: REAL := 10.0; // Distance from mast slide full extension.
	
	(* ----------------------- SCREW MODE: Leave/return to drive ------------------------ *)
	RETURNING_TO_DRIVE: BOOL := FALSE;
	UC_RETURN_POS: REAL;
	
	(* ----------------------- SCREW MODE: UR stall detect ------------------------------ *)
	// This flag is set false at the beginning of every screw drive, then true when we have stalled
	//	and tne controls has attempted the stall recovery.
	UR_STALL_RECOVERY: BOOL := FALSE;
	// The furthest the tip of the drill has been in the ground during a stalled screw drive.  Used so that
	//	after the drill has been pulled up to try to protect it when we re-engage with the ground.
	UR_STALL_FURTHEST_EXTENT: REAL;
	
	(* ---------------------- SCREW MODE: LC stall detect ---------------------- *)
	// Time when the LC velocity dropped low enough that we suspect a stall.
	LC_STALL_START: REAL := 0;
	LC_STALL_SUSPECTED: BOOL := FALSE;
	LC_RAMPUP: BOOL := FALSE;
	
	(* ---------------------- RWP MODE STATES and DATA HERE ---------------------- *)
	RWP_STATE: eRWPStates;
	RWP_MODE_STATE_CHANGE: BOOL := FALSE;
	RWP_MODE_PAUSED: BOOL := FALSE;
	RWP_MODE_PAUSED_CHANGE: BOOL := FALSE;

	YAW_SQUARE_TO_LASER: REAL := 0.0;

	(* ---------------------- MISCELLANEOUS STATE DATA ---------------------- *)
	TARGET_PLATE_UP: BOOL := FALSE;
	
	(* ----------------------- TOP LEVEL FBs -------------------------------------------- *)
	(*
	processRemote_01: processRemote;
	machineState_01: machineState;
	runActuators_01: runActuators;
	xyzTrueMotion_01: xyzTrueMotion;
	*)
	
END_VAR

// SafetyPLC/Application/PLC_PRG
PROGRAM PLC_PRG
VAR
END_VAR

END_PROGRAM

// StandardPLC/Application/POUs/PLC_PRG
PROGRAM PLC_PRG
VAR
	TMP: INT;
	ON: INT;
	OFF: INT;
	CYCLE: TON;
	NEEDS_INIT: BOOL := TRUE;
	GPS_1: GPS;
	
	// sys time
	US_TIME: DWORD;
	US: SysTime;
	US_TIME_LAST: DWORD := 0;
	US_START: DWORD := 0;
END_VAR


TMP := TMP + 1;

US_TIME_LAST := US_TIME;
SysTimeGetUs(pUsTime := US);
US_TIME := ULINT_TO_DWORD(US);

CYCLE(IN := NOT CYCLE.Q, PT := T#5S);

IF NEEDS_INIT THEN
	NEEDS_INIT := FALSE;
	//CheckSumTest();
	//Enum();
	//DeRef();
	//Type_conversions();
	//SineCheck();
	//DivByZero ();
	//PointerMath();
	//CheckSumTest();
	//ArrayConversionTest();
	//CheckForExtendedCAN();
	//ConvertRealToCAN();
	//UnderstandingDataTypes();
	//Timing();
	//ProfileCheck();
	//Test_Data_Averaging();
	//CoordinateTransforms();
	//XdjustNxtSiMMotor();
	//MiscChecks();
	//GPS();
	Parsing();
END_IF

//TD_SIM();
//UnderstandingDataTypes();
//LogicalOperators();
//CheckUDINTdeconstruction();
//ArrayConstruction();
//TdActuatorMoves();
//Test_Data_Averaging();
//CoordinateTransforms();
//ArrayConversionTest();
//DivByZero();
//ProfileCheck();
GPS_1();
//Timing();
//ConvertCanToText();
//ddtLayers();
//();
pnezD_decoding();
//DynamicList();
Arrays();

IF CYCLE.Q THEN
	ON := ON + 1;
ELSE
	OFF := OFF + 1;
END_IF

END_PROGRAM

// StandardPLC/Application/POUs/Type_conversions
PROGRAM Type_conversions
VAR
	Var1: STRING;
	Var2: STRING;
	Var3: STRING;
	Var4: STRING;
	sVar1: STRING;
	sVar2: STRING;

	iVar1: STRING;
	infoVar1: __SYSTEM.VAR_INFO;
	infoVar2: __SYSTEM.VAR_INFO;

			
	test1 : INT;
	test2 : INT;
	test3 : INT;
	test4 : INT;

		WIRED_OUTS: ARRAY [1..4] OF POINTER TO INT :=
	[
		ADR(test1),       //1
		ADR(test2),       //2
		ADR(test3),       //3
		ADR(test4)        //4

	];
	
	
END_VAR

test1 := 11;
test2 := 22;
test3 := 33;

Var1 := TO_STRING(test1);
infoVar1 := __VARINFO(test1);
sVar1 := infoVar1.Symbol;

Var3 := TO_STRING(WIRED_OUTS[1]^);
infoVar2 := __VARINFO(WIRED_OUTS[1]^);
sVar2 := infoVar2.Symbol;

END_PROGRAM

// StandardPLC/Application/POUs/GPS/GPS
FUNCTION_BLOCK GPS
VAR_INPUT
END_VAR
VAR_OUTPUT
END_VAR

VAR
	INIT: BOOL := TRUE;
	// GPS data - targets to address heading, x, y, z offsets
	
	GPS_WP_AUTOTARGET: BOOL := FALSE;

	(*
		0: not used	
		1: not all selected axes in range to autotarget;
		2: all selected axes in range to autotarget;
		3: all axes on target
	*)
	GPS_AUTOTARGET_STATUS_CHECK: UINT := 0; 
	(*
	YAW_SETTLED_IN_BAND: GPS_SETTLED_WITHIN_BAND_1S;
	Y_SETTLED_IN_BAND: GPS_SETTLED_WITHIN_BAND_1S; *)
	i: INT;
	GpsUpdate: GpsUpdate;
END_VAR

(*processes GPS input
	inputs:
	- gps offsets
	- axes autotargeting selection
	outputs:
	- whether actuators should auto-move using gps
	- when actuators are on target
	other functions:
	- sets limits for autotarget to be enabled within
*)
//(*
IF INIT THEN // initiate gps axes
	(*
	FOR i := 1 TO NUM_GPS_AXES DO
		configGPSaxis(i, GPS_RANGE_ARRAY[i], GPS_TARGET_TOLERANCE[i]);
	END_FOR;
	//*)
	GPS_AXES[GPS_HEADING].AXIS_RANGE_MAX := 24;
	GPS_AXES[GPS_HEADING].AXIS_RANGE_MIN := -24;
	GPS_AXES[GPS_X].AXIS_RANGE_MAX := 30;
	GPS_AXES[GPS_X].AXIS_RANGE_MIN := 0;
	GPS_AXES[GPS_Y].AXIS_RANGE_MAX := 24;
	GPS_AXES[GPS_Y].AXIS_RANGE_MIN := -24;
	GPS_AXES[GPS_Z].AXIS_RANGE_MAX := 167.5;
	GPS_AXES[GPS_Z].AXIS_RANGE_MIN := 2;
	//TD_SIM(INIT := INIT);
	TD_SIM(INIT);
END_IF
//*)

// apply simulation values to GPS_AXES
FOR i := 1 TO 4 DO
	GPS_AXES[i].OFFSET := GPS_SIM_OFFSETS[i];
END_FOR
GpsUpdate(INIT := INIT); // update status for all gps axes
GpsAutotargetInRange(GPS_RANGE_MARGIN);
//AND GPS_RTK_SIGNAL_DELAY < GPS_RTK_SIGNAL_CRITICAL_LIMIT  // activate once we can access this information over CAN - waiting on StonEx software update

// check for settled within band
(*
IF ( RWP_STATE = RWP_STATE_SQUARE_YAW ) AND AUTOMATIC THEN
	YAW_SETTLED_IN_BAND( INIT := isRwpModeStateChange(), GPS_AXIS := GPS_HEADING );
END_IF
*)

GPS_AUTOTARGET_STATUS_CHECK := 4; 
FOR i := 1 TO NUM_GPS_AXES DO
	IF GPS_AXES[i].AUTOTARGET_ON THEN
		// check if any status is less than in range or on target and reduce to lowest common denominator:
		(* Range status:
		0: not in range to auto-target; 
		1: in range to move to target but not on target, OR autotarget not selected;
		2: in range to move to target, not on target; 
		3: within target specification; 
		*)
		GPS_AUTOTARGET_STATUS_CHECK := MIN(GPS_AUTOTARGET_STATUS_CHECK, GPS_AXES[i].RANGE_STATUS);
	END_IF
END_FOR

(* GPS_AUTOTARGET_STATUS by bit#:
	0: AUTOTARGET engaged
	1-4: selected axis engaged
	10: all gps axes are in range for autotarget
	11: all gps axes are on target
*)
(*
GPS_AUTOTARGET_STATUS.ALL_GPS_AXES_IN_RANGE := (GPS_AUTOTARGET_STATUS_CHECK > 1) ; 
GPS_AUTOTARGET_STATUS.ALL_GPS_AXES_ON_TARGET := (GPS_AUTOTARGET_STATUS_CHECK > 2) ; 
*)
INIT := FALSE;

(*
GpsAutoTrack(X_OFFSET_BEGIN := GPS_AXES[GPS_X].OFFSET, Y_OFFSET_BEGIN := GPS_AXES[GPS_Y].OFFSET, 
			 YAW_OFFSET_BEGIN := GPS_AXES[GPS_HEADING].OFFSET, Z_OFFSET_BEGIN := GPS_AXES[GPS_Z].OFFSET) ;
			 *)

GpsAutoTrack(X_OFFSET_BEGIN := GPS_AXES[GPS_X].OFFSET, Y_OFFSET_BEGIN := GPS_AXES[GPS_Y].OFFSET, YAW_OFFSET_BEGIN := GPS_AXES[GPS_HEADING].OFFSET,
			LEFT_TRACK_OUTPUT_MAGNITUDE => GPS_LEFT_JS, RIGHT_TRACK_OUTPUT_MAGNITUDE => GPS_RIGHT_JS, 
			LEFT_TRACK_OUTPUT_POSITIVE => GPS_LEFT_POSITIVE, RIGHT_TRACK_OUTPUT_POSITIVE => GPS_RIGHT_POSITIVE);
			
//BoundAxes();

END_FUNCTION_BLOCK

// StandardPLC/Application/POUs/GPS/TD_SIM
FUNCTION TD_SIM
VAR_INPUT
	INIT: BOOL := TRUE;
	
END_VAR

IF INIT THEN
	INIT := FALSE;
	AXES[AXIS_BOOM_SWING].FEEDBACK.POSITION_ENGR := 0;
	AXES[AXIS_X_SLIDE].FEEDBACK.POSITION_ENGR := 15;
	AXES[AXIS_YAW].FEEDBACK.POSITION_ENGR := 0;
	AXES[AXIS_Z_SLIDE].FEEDBACK.POSITION_ENGR := 100;
	
END_IF

END_FUNCTION

// StandardPLC/Application/POUs/GPS/GpsUpdate
FUNCTION_BLOCK GpsUpdate
	(* Range status:
		0: not in range to auto-target; 
		1: in range to move to target but not on target, OR autotarget not selected;
		2: in range to move to target, not on target; 
		3: within target specification; 
		*)

VAR_INPUT
	INIT: BOOL := TRUE;
END_VAR
VAR
	i: INT := 0;
	AUTOTARGET_WORD: WORD := 0;
	GPS_FIXED: boxcarFilter;
	
	GPS_RTK_FIXED_DATA_POINTS: ARRAY [1..25] OF REAL := [25(0)];
	GPS_FIXED_FILTERED: REAL := 0;
	GPS_FIXED_FILTER_VALID: BOOL := FALSE;
	
	GPS_FIXED_FILTER_COUNTER: USINT := 0; // use to time when to send data
	GPS_FIXED_FILTER_SAMPLE_TIMER: TON;
	GPS_INIT: BOOL := TRUE;
	
END_VAR

IF INIT THEN
	INIT := FALSE;
	FOR i := 1 TO NUM_GPS_AXES DO
		GPS_AXES[i].OFFSET := GPS_SIM_OFFSETS[i];
	END_FOR
END_IF

FOR i := 1 TO NUM_GPS_AXES DO
	
	GPS_AXES[i].REACH := GPS_SETTINGS[i, GPS_AXIS_IN_RANGE];
	GPS_AXES[i].TARGET_LIMIT := GPS_SETTINGS[i, GPS_AXIS_ON_TARGET];
	
	IF (ABS(GPS_AXES[i].OFFSET) < GPS_AXES[i].TARGET_LIMIT) THEN
		GPS_AXES[i].RANGE_STATUS := TO_UINT(GPS_AXIS_ON_TARGET);
	ELSIF (ABS(GPS_AXES[i].OFFSET) < GPS_AXES[i].REACH) THEN
		GPS_AXES[i].RANGE_STATUS := TO_UINT(GPS_AXIS_IN_RANGE);
	ELSIF (ABS(GPS_AXES[i].OFFSET) < GPS_AXES[i].REACH) OR (NOT GPS_AXES[i].AUTOTARGET_ON) THEN
		GPS_AXES[i].RANGE_STATUS := TO_UINT(GPS_AXIS_NOT_IN_RANGE_NOT_IN_AUTO);
	ELSE
		GPS_AXES[i].RANGE_STATUS := TO_UINT(GPS_AXIS_NOT_IN_RANGE);
	END_IF

	AUTOTARGET_WORD := TO_WORD (SHR(GPS_AUTOTARGET_SELECTION, i)); 
	GPS_AXES[i].AUTOTARGET_ON := AUTOTARGET_WORD.0; // update whether axis is selected for autotarget
	
END_FOR

//IF MACHINE_MODE = RWP_MODE THEN
	GpsTdToWorldFixedYaw( X_TD_WP := GPS_AXES[GPS_X].OFFSET, Y_TD_WP := GPS_AXES[GPS_Y].OFFSET, YAW_BEGIN := GPS_AXES[GPS_HEADING].OFFSET, 
		X_WORLD_WP => GPS_AXES[GPS_X].OFFSET_WORLD_FRAME, Y_WORLD_WP =>  GPS_AXES[GPS_Y].OFFSET_WORLD_FRAME);
//END_IF
GpsTdToWorldFixAll2d( X_OFFSET_BEGIN := GPS_SIM_OFFSETS[GPS_X], Y_OFFSET_BEGIN :=  GPS_SIM_OFFSETS[GPS_Y], 
						YAW_OFFSET_BEGIN := GPS_SIM_OFFSETS[GPS_HEADING], Z_OFFSET_BEGIN := GPS_SIM_OFFSETS[GPS_Z]);

debug[2] := debug[2] + 1;

(*
IF GPS_VENDOR_VALUE > 0 THEN
	GPS_FIXED_FILTER_SAMPLE_TIMER(IN := NOT GPS_FIXED_FILTER_SAMPLE_TIMER.Q, PT := T#200MS); // 5 Hz sampling
	IF GPS_INIT THEN
		GPS_FIXED(INIT := TRUE, READING := TO_REAL(GPS_RTK_FIXED), 
			SAMPLES := GPS_RTK_FIXED_DATA_POINTS, FILTERED => GPS_FIXED_FILTERED, VALID => GPS_FIXED_FILTER_VALID);
		GPS_INIT := FALSE;
	END_IF
	IF GPS_FIXED_FILTER_SAMPLE_TIMER.Q THEN
		GPS_FIXED(INIT := FALSE, READING := TO_REAL(GPS_RTK_FIXED), 
			SAMPLES := GPS_RTK_FIXED_DATA_POINTS, FILTERED => GPS_FIXED_FILTERED, VALID => GPS_FIXED_FILTER_VALID);
		
	END_IF
	IF GPS_FIXED_FILTERED > 0.9 THEN // allows 2 falses in 25 samples, or 92%  Should this be higher?
		GPS_AUTOTARGET_STATUS.GPS_STABLE_5S := TRUE;
		debug_ctr_4 := debug_ctr_4 + 1;
	ELSE
		GPS_AUTOTARGET_STATUS.GPS_STABLE_5S := FALSE;
		debug_ctr_5 := debug_ctr_5 + 1;
	END_IF
	GPS_READY := GPS_FIXED_FILTER_VALID AND (GPS_HRMS <= GPS_MIN_HRMS) AND (GPS_VRMS < GPS_MIN_VRMS) AND GPS_AUTOTARGET_STATUS.GPS_STABLE_5S; //
END_IF
*)

END_FUNCTION_BLOCK

// StandardPLC/Application/POUs/GPS/GpsTdToWorldFixedYaw
FUNCTION GpsTdToWorldFixedYaw : REAL // only considers rotating at yaw pivot

VAR_INPUT
	X_TD_WP: REAL := 0; // offsets from WP given by gps, + is forward of operator 
	Y_TD_WP: REAL := 0; // + is to the right of operator (facing forward at rear [mast end] of TD)
	YAW_BEGIN: REAL := 0; // heading offset to rotate by as given by gps, + is moving mast to the right (CCW) of operator
END_VAR
VAR_OUTPUT
	X_WORLD_WP: REAL :=0; // final x from WP after yaw move to align yaw arm with North-South, + forward of operator 
	Y_WORLD_WP: REAL :=0; // final y from WP after yaw move, + to operators right
END_VAR

(* 
take gps offsets that are given in reference to wp and:
 a) translate them to yaw pivot
 b) rotate them by yaw offset
 c) translate back to wp in new reference frame
 
 This gives us the angle we need to rotate yaw arm by and the new y and x offsets to the target point after rotating the arm
*)

// X_TD_WP  - 135;  translate origin from wp to yaw pivot
// Y_TD_WP; doesn't change for translation along 
RotateGpsTdToWorldNS( X_TD := X_TD_WP - (YAW_PIVOT_TO_DRILL_ROD + AXES[AXIS_X_SLIDE].FEEDBACK.POSITION_ENGR), Y_TD := Y_TD_WP, YAW_BEGIN := YAW_BEGIN, X_WORLD => X_WORLD_WP, Y_WORLD => Y_WORLD_WP);
X_WORLD_WP := X_WORLD_WP + YAW_PIVOT_TO_DRILL_ROD + AXES[AXIS_X_SLIDE].FEEDBACK.POSITION_ENGR; // translate origin from wp to yaw pivot
// Y_WORLD_WP doesn't change for translation along x

END_FUNCTION

// StandardPLC/Application/POUs/GPS/RotateGpsTdToWorldNS
FUNCTION RotateGpsTdToWorldNS : REAL // input offsets in reerence to yaw pivot, outputs offsets after given rotation
VAR_INPUT
	X_TD: REAL := 0; // offsets given by gps, + is forward of operator 
	Y_TD: REAL := 0; // + is to the right of operator (facing forward at rear [mast end] of TD)
	YAW_BEGIN: REAL := 0; // heading offset to rotate by as given by gps, + is moving mast to the right (CCW) of operator
END_VAR
VAR_OUTPUT
	X_WORLD: REAL :=0; // final x after yaw move to align yaw arm with North-South, + forward of operator 
	Y_WORLD: REAL :=0; // final y after yaw move, + to operators right
END_VAR
VAR
END_VAR


X_WORLD := X_TD * COS_DEG(YAW_BEGIN) - Y_TD * SIN_DEG(YAW_BEGIN); // rotate origin at yaw pivot by gps heading offset
Y_WORLD := X_TD * SIN_DEG(YAW_BEGIN) + Y_TD * COS_DEG(YAW_BEGIN);

END_FUNCTION

// StandardPLC/Application/POUs/Utilities/Conversions/COS_DEG
FUNCTION COS_DEG : REAL
VAR_INPUT
	DEGREES: REAL;
END_VAR
VAR
	RADIANS: REAL;
END_VAR


//RADIANS := (3.14159 * DEGREES / 180.0);
//RADIANS := (3.14159265359 * DEGREES / 180.0);
RADIANS := (Pi * DEGREES / 180.0);
COS_DEG := COS(RADIANS);

END_FUNCTION

// StandardPLC/Application/POUs/Utilities/Conversions/SIN_DEG
FUNCTION SIN_DEG: REAL
VAR_INPUT
	DEGREES: REAL;
END_VAR
VAR
	RADIANS: REAL;
END_VAR

//RADIANS := (3.14159 * DEGREES / 180.0);
//RADIANS := (3.14159265359 * DEGREES / 180.0);
RADIANS := (Pi * DEGREES / 180.0);
SIN_DEG := SIN(RADIANS);

END_FUNCTION

// StandardPLC/Application/POUs/GPS/GpsTdToWorldFixAll2d
// calculations confirmed via SolidWorks

FUNCTION GpsTdToWorldFixAll2d : REAL // bring back to boom swing pivot

VAR_INPUT
	X_OFFSET_BEGIN: REAL := 0; // offsets from WP given by gps, in TD frame, + is forward of operator 
	Y_OFFSET_BEGIN: REAL := 0; // + is to the right of operator (facing forward at rear [mast end] of TD)
	YAW_OFFSET_BEGIN: REAL := 0; // heading offset to rotate by as given by gps, + is moving mast to the right (CCW) of operator
	Z_OFFSET_BEGIN: REAL := 0; // + is up
	
	// X_TD_WP: REAL := 0; // offsets from WP given by gps, in TD frame, + is forward of operator 
	// Y_TD_WP: REAL := 0; // + is to the right of operator (facing forward at rear [mast end] of TD)
END_VAR
VAR
	(*
	BS_ANGLE_NS_DELTA: REAL := 0;
	BS_ANGLE_WORLD_NS: REAL := 0;
	BS_ANGLE_NS_TO_Y_TARGET_DELTA: REAL := 0;
	
	X_OFFSET: REAL := 0; // offsets from WP given by gps, in TD frame, + is forward of operator 
	Y_OFFSET: REAL := 0; // + is to the right of operator (facing forward at rear [mast end] of TD)
	YAW_OFFSET: REAL := 0; // heading offset to rotate by as given by gps, + is moving mast to the right (CCW) of operator
	//*)
	YAW_PIVOT_TO_DRILL_ROD: REAL := 135; //TD3
	
	
END_VAR

VAR_OUTPUT
	(*
	BS_TARGET: REAL := 0;
	X_SLIDE_TARGET: REAL := 0;
	YAW_TARGET: REAL := 0;
	*)
	(*
	X_YAW_PIVOT_TO_TARGET_ORIGINAL: REAL := 0; // X from yaw pivot to target before rotation at yaw pivot
	Y_YAW_PIVOT_TO_TARGET_ORIGINAL: REAL := 0; // Y from yaw pivot to target before rotation at yaw pivot
	X_YAW_PIVOT_TO_TARGET_ROTATED_AT_YAW_PIVOT: REAL := 0; // X from yaw pivot to target after rotation to bs frame at yaw pivot
	Y_YAW_PIVOT_TO_TARGET_ROTATED_AT_YAW_PIVOT: REAL := 0; // Y from yaw pivot to target after rotation to bs frame at pivot
	X_BS_PIVOT_TO_TARGET_ORIGINAL: REAL := 0; // X from bs pivot to target before rotation at bs pivot
	Y_BS_PIVOT_TO_TARGET_ORIGINAL: REAL := 0; // Y from bs pivot to target before rotation at bs pivot
	X_BS_PIVOT_TO_TARGET_ROTATED_AT_YAW_PIVOT: REAL := 0; // X from bs pivot to target after rotation at bs pivot
	Y_BS_PIVOT_TO_TARGET_ROTATED_AT_YAW_PIVOT: REAL := 0; // Y from bs pivot to target after rotation at bs pivot
	
	
	X_BS_TARGET: REAL := 0; // final x from WP after yaw move to align yaw arm with North-South, + forward of operator 
	Y_BS_TARGET: REAL := 0; // final y from WP after yaw move, + to operators right
	X_WORLD_WP: REAL := 0; // final x from WP after yaw move to align yaw arm with North-South, + forward of operator 
	Y_WORLD_WP: REAL := 0; // final y from WP after yaw move, + to operators right
	*)
END_VAR

X_OFFSET_BEGIN := X_OFFSET_BEGIN/10; // convert mm to cm
Y_OFFSET_BEGIN :=  Y_OFFSET_BEGIN/10; // convert mm to cm
//YAW_OFFSET_BEGIN := YAW_OFFSET_BEGIN;
Z_OFFSET_BEGIN := Z_OFFSET_BEGIN/10; // convert mm to cm
YAW_ARM_LENGTH := YAW_PIVOT_TO_DRILL_ROD + AXES[AXIS_X_SLIDE].FEEDBACK.POSITION_ENGR;
//(* 
// * WP frame - origin at WP *
//  (if 3d have to first rotate at wp to get pitch and roll aligned with yaw arm)
// 1) translate origin to reference yaw pivot (translation)

X_OFFSETS[1] := X_OFFSET_BEGIN - YAW_ARM_LENGTH;;
Y_OFFSETS[1] := Y_OFFSET_BEGIN;

// * WP frame - origin at yaw pivot *
// 2) rotate origin at yaw pivot to match bs frame (rotation)
// YAW_ROTATION := AXES[AXIS_YAW].FEEDBACK.POSITION_ENGR; // offset from Boom Swing

X_OFFSETS[2] := X_OFFSETS[1] * COS_DEG(AXES[AXIS_YAW].FEEDBACK.POSITION_ENGR) - Y_OFFSETS[1] * SIN_DEG(AXES[AXIS_YAW].FEEDBACK.POSITION_ENGR); // rotate origin at yaw pivot by gps heading offset
Y_OFFSETS[2] := X_OFFSETS[1] * SIN_DEG(AXES[AXIS_YAW].FEEDBACK.POSITION_ENGR) + Y_OFFSETS[1] * COS_DEG(AXES[AXIS_YAW].FEEDBACK.POSITION_ENGR);

// * BS frame - origin AT yaw pivot *
// 3) translate origin to bs pivot

X_OFFSETS[3] := X_OFFSETS[2] - BS_LENGTH;;
Y_OFFSETS[3] := Y_OFFSETS[2];

// * BS frame - origin at BS pivot *
// 4) rotate origin at bs pivot to world frame
//	- rotate by BS_ANGLE_NS_DELTA
BS_ANGLE_NS_DELTA := YAW_OFFSET_BEGIN + -1 * AXES[AXIS_YAW].FEEDBACK.POSITION_ENGR; //(Yaw is opposite sign)
BS_ANGLE_WORLD_NS := BS_ANGLE_NS_DELTA + AXES[AXIS_BOOM_SWING].FEEDBACK.POSITION_ENGR;

X_OFFSETS[4] := X_OFFSETS[3] * COS_DEG(BS_ANGLE_NS_DELTA) - Y_OFFSETS[3] * SIN_DEG(BS_ANGLE_NS_DELTA); // rotate origin at yaw pivot by gps heading offset
Y_OFFSETS[4] := X_OFFSETS[3] * SIN_DEG(BS_ANGLE_NS_DELTA) + Y_OFFSETS[3] * COS_DEG(BS_ANGLE_NS_DELTA);

// * WORLD frame - origin at BS pivot *
// 5) calculate bs angle to move BS by to get WORLD_Y to 0 in WORLD frame      																** MOVE BS **
BS_ANGLE_NS_TO_Y_TARGET_DELTA := ASIN_DEG ( Y_OFFSETS[4] / BS_LENGTH );
TARGET_POSITIONS_METHOD_2[GPS_Y]  := BS_ANGLE_WORLD_NS + BS_ANGLE_NS_TO_Y_TARGET_DELTA;
// 6) move origin to yaw pivot: translate in x and y (and z if 3d) to move origin to yaw pivot (translation)
// - x translation := COS_DEG ( BS_ANGLE_NS_TO_Y_TARGET_DELTA ) * BS_LENGTH
X_OFFSETS[5] := X_OFFSETS[4] + COS_DEG ( BS_ANGLE_NS_TO_Y_TARGET_DELTA ) * BS_LENGTH;
// y translation := SIN_DEG ( BS_ANGLE_NS_TO_Y_TARGET_DELTA ) * BS_LENGTH
Y_OFFSETS[5] := Y_OFFSETS[4] - SIN_DEG ( BS_ANGLE_NS_TO_Y_TARGET_DELTA ) * BS_LENGTH; // y offset should = 0 at this point

// * WORLD frame - origin at yaw pivot *
// 7) rotate yaw to align with world NS 													

YAW_OFFSETS[1] := YAW_OFFSET_BEGIN - ( TARGET_POSITIONS_METHOD_2[GPS_Y] - AXES[AXIS_BOOM_SWING].FEEDBACK.POSITION_ENGR );

TARGET_POSITIONS_METHOD_2[GPS_HEADING] := -1 * YAW_OFFSETS[1] + AXES[AXIS_YAW].FEEDBACK.POSITION_ENGR; //original heading offset + bs move		** MOVE YAW **

(* don't do this because coordinates are already in world frame.  Just translate along yaw arm to wp
X_OFFSETS[6] := X_OFFSETS[5] * COS_DEG(BS_ANGLE_NS_DELTA) - Y_OFFSETS[5] * SIN_DEG(BS_ANGLE_NS_DELTA); // rotate origin at yaw pivot by gps heading offset
Y_OFFSETS[6] := X_OFFSETS[5] * SIN_DEG(BS_ANGLE_NS_DELTA) + Y_OFFSETS[5] * COS_DEG(BS_ANGLE_NS_DELTA);
*)

// 8) translate origin from yaw pivot to wp

X_OFFSETS[6] := X_OFFSETS[5] + YAW_ARM_LENGTH;;
Y_OFFSETS[6] := Y_OFFSETS[5];


// * WORLD frame - origin at WP * 
// 9) move x-slide to put WP at 0 x
TARGET_POSITIONS_METHOD_2[GPS_X] := AXES[AXIS_X_SLIDE].FEEDBACK.POSITION_ENGR + ( -1 * X_OFFSETS[6]);	// x-slide moves opposite direction of offset
// * WORLD frame - origin at WP * * WP frame - origin AT WP * ( should be the same now )													** MOVE X-SLIDE **
 
// get z_slide 2d
TARGET_POSITIONS_METHOD_2[GPS_Z] := AXES[AXIS_Z_SLIDE].FEEDBACK.POSITION_ENGR + Z_OFFSET_BEGIN;	// 											** MOVE Z-SLIDE **			
 
//*)




(*
// Y_TD_WP; doesn't change for translation along 
ROTATE_DEG_FROM_YAW_TO_BS := -AXES[AXIS_YAW].FEEDBACK.POSITION_ENGR;

// TRANSLATE ORIGIN FROM WP TO YAW PIVOT (Y doesn't change in this translation)
X_YAW_PIVOT_TO_TARGET_ORIGINAL := X_TD_WP - 135;
Y_YAW_PIVOT_TO_TARGET_ORIGINAL := Y_TD_WP;

// ROTATE ABOUT YAW PIVOT FROM YAW ARM FRAME TO BOOM SWING FRAME
RotateGpsTdToWorldNS( X_TD := X_YAW_PIVOT_TO_TARGET_ORIGINAL, Y_TD := Y_YAW_PIVOT_TO_TARGET_ORIGINAL, YAW_BEGIN := ROTATE_DEG_FROM_YAW_TO_BS,
					  X_WORLD => X_YAW_PIVOT_TO_TARGET_ROTATED_AT_YAW_PIVOT, Y_WORLD => Y_YAW_PIVOT_TO_TARGET_ROTATED_AT_YAW_PIVOT );
					  
// In BS frame now, so MOVE TO ORIGIN OF BS
X_BS_PIVOT_TO_TARGET_ORIGINAL := X_YAW_PIVOT_TO_TARGET_ROTATED_AT_YAW_PIVOT - 135; // X from bs pivot to target before rotation at bs pivot
Y_BS_PIVOT_TO_TARGET_ORIGINAL := Y_YAW_PIVOT_TO_TARGET_ROTATED_AT_YAW_PIVOT; // Y from bs pivot to target before rotation at bs pivot

// ROTATE FROM BS FRAME TO WORLD FRAME

					  
//X_WORLD_WP := X_WORLD_WP + 135; // translate origin from yaw pivot to wp

// GET BS MOVE to cancel y offset,

// GET X OFFSET after BS move	



			  
// TRANSLATE TO BS ORIGIN THEN ROTATE TO WORLD FRAME

// Y_WORLD_WP doesn't change for translation along x
//*)

END_FUNCTION

// StandardPLC/Application/POUs/Utilities/Conversions/ASIN_DEG
FUNCTION ASIN_DEG: REAL
VAR_INPUT
	VALUE: REAL;
END_VAR
VAR
END_VAR

// ASIN_DEG := (180 * ASIN(VALUE)) / 3.14159;

IF ABS(VALUE) > 1 THEN // prevent killing PLC with a NaN if bad value sent
	VALUE := MAX(MIN(VALUE, -1),1);
END_IF

ASIN_DEG := (180 * ASIN(VALUE)) / Pi;

END_FUNCTION

// StandardPLC/Application/POUs/GPS/GpsAutotargetInRange
FUNCTION GpsAutotargetInRange : BOOL

VAR_INPUT
	PERCENT_MARGIN: REAL;
END_VAR
VAR
	
	i: USINT := 0;
	//PERCENT_MARGIN_AS_FACTOR: REAL;
	
	X_DELTA_FROM_BS_MOVE: REAL := 0;
END_VAR

// return whether gps is in range of actuators
// multiply offset by ( 1 + PERCENT_MARGIN )
// if target ( current position + offset ): min < target < max then good

GpsAutotargetInRange := TRUE; // Start true, any failure turns it false
PERCENT_MARGIN_AS_FACTOR := 1 - ( PERCENT_MARGIN / 100 );
FOR i := 0 TO 4 DO
	GPS_IN_RANGE[i] := FALSE;
END_FOR

// bs range: +/- 25 deg
//(*
TARGET_POSITIONS_METHOD_1[GPS_Y] := GPS_Y_TO_BS_ANGLE( AXES[AXIS_YAW].FEEDBACK.POSITION_ENGR, GPS_AXES[GPS_HEADING].OFFSET, 
						GPS_AXES[GPS_X].OFFSET_WORLD_FRAME/10, GPS_AXES[GPS_Y].OFFSET_WORLD_FRAME/10 ) // convert mm to cm
						+ AXES[AXIS_BOOM_SWING].FEEDBACK.POSITION_ENGR;
 
IF 	ABS(TARGET_POSITIONS_METHOD_1[GPS_Y]) > PERCENT_MARGIN_AS_FACTOR * 24 THEN
	GpsAutotargetInRange := FALSE;
ELSE
  	GPS_IN_RANGE[GPS_Y] := 1;
END_IF
//*)

// x slide range: 0-30 cm
//(*
// convert offset to cm, and moving fwd is (- to 0) for actuator
X_DELTA_FROM_BS_MOVE := -1 * ( ( BS_LENGTH ) - 
						TO_REAL ( SQRT ( EXPT ( BS_LENGTH, 2 ) - EXPT ( GPS_AXES[GPS_Y].OFFSET_WORLD_FRAME/10, 2 ) ) ) ); // switch signs to get offset
TARGET_POSITIONS_METHOD_1[GPS_X] := AXES[AXIS_X_SLIDE].FEEDBACK.POSITION_ENGR - ( GPS_AXES[GPS_X].OFFSET_WORLD_FRAME / 10 + X_DELTA_FROM_BS_MOVE );

IF 	( TARGET_POSITIONS_METHOD_1[GPS_X] > PERCENT_MARGIN_AS_FACTOR * 30 ) 
	OR ( TARGET_POSITIONS_METHOD_1[GPS_X] < (  0 + ( 1 - PERCENT_MARGIN_AS_FACTOR ) * 30 ) )
	THEN
	GpsAutotargetInRange := FALSE;
ELSE
  	GPS_IN_RANGE[GPS_X] := 1;
END_IF
//*)

// yaw range: +/- xx deg
(*
 TARGET_POS := GPS_Y_TO_BS_ANGLE( AXES[AXIS_YAW].FEEDBACK.POSITION_ENGR, GPS_AXES[GPS_HEADING].OFFSET, 
							GPS_AXES[GPS_X].OFFSET_WORLD_FRAME, GPS_AXES[GPS_Y].OFFSET_WORLD_FRAME ) - GPS_AXES[GPS_HEADING].OFFSET
							+ AXES[AXIS_YAW].FEEDBACK.POSITION_ENGR; // (-) heading offset and (+) boom swing angle because yaw is reversed
							*)
TARGET_POSITIONS_METHOD_1[GPS_HEADING] := GPS_Y_TO_BS_ANGLE( AXES[AXIS_YAW].FEEDBACK.POSITION_ENGR, GPS_AXES[GPS_HEADING].OFFSET, 
							GPS_AXES[GPS_X].OFFSET_WORLD_FRAME/10, GPS_AXES[GPS_Y].OFFSET_WORLD_FRAME/10 ) - GPS_AXES[GPS_HEADING].OFFSET
							+ AXES[AXIS_YAW].FEEDBACK.POSITION_ENGR; // (-) heading offset and (+) boom swing angle because yaw is reversed
IF 	ABS(TARGET_POSITIONS_METHOD_1[GPS_HEADING]) > PERCENT_MARGIN_AS_FACTOR * 24 THEN
	GpsAutotargetInRange := FALSE;
ELSE
  	GPS_IN_RANGE[GPS_HEADING] := 1;
END_IF

// Z slide range: 5 - xx cm
TARGET_POSITIONS_METHOD_1[GPS_Z] := GPS_AXES[GPS_Z].OFFSET / 10 + AXES[AXIS_Z_SLIDE].FEEDBACK.POSITION_ENGR; // convert mm to cm
IF 	TARGET_POSITIONS_METHOD_1[GPS_Z] > PERCENT_MARGIN_AS_FACTOR * 167.5 
	OR TARGET_POSITIONS_METHOD_1[GPS_Z] < ( 2 + ( ( PERCENT_MARGIN / 100 ) * 167.5 ) ) 
	THEN
	GpsAutotargetInRange := FALSE;
	debug[4] := debug[4] + 1;
ELSE
  	GPS_IN_RANGE[GPS_Z] := 1;
	debug[5] := debug[5] + 1000;
END_IF

GPS_IN_RANGE[0] := GpsAutotargetInRange;

debug[3] := debug[3] + 1;

END_FUNCTION

// StandardPLC/Application/POUs/GPS/GPS_Y_TO_BS_ANGLE
// angle to move BS by to align end of BS (yaw pivot) with y of target
// input offsets and yaw angle as given by gps and td respectively
// THIS ONE WORKS - only difference is Y_DELTA_WORLD in td code is /10 to convert mm to cm

FUNCTION GPS_Y_TO_BS_ANGLE : REAL 

VAR_INPUT // most of these will be available in TD code
	YAW_ANGLE: REAL; // angle of yaw arm relative to BS per TD
	HEADING_OFFSET_GPS: REAL; // YAW_BEGIN, or heading offset of wp in world; + is moving mast to the right (CCW) of operator
	X_TD_WP: REAL := 0; // x offset from WP as given by gps, + is forward of operator 
	Y_TD_WP: REAL := 0; // + is to the right of operator (facing forward at rear [mast end] of TD)
	
END_VAR
VAR
	BS_ANGLE_WORLD: REAL; //  Angle in world terms (not offset - ccw is positive)
	BS_LENGTH: REAL := 135; // length of boom swing arm
	BS_PIVOT_TO_YAW_PIVOT_Y_WORLD: REAL; // Y delta of BS arm in world frame from bs pivot to yaw pivot
	BS_PIVOT_TO_TARGET_Y_DELTA: REAL; // distance in Y from BS origin (bs pivot) to target point
	BS_PIVOT_TO_TARGET_Y_HEADING: REAL; // BS angle from pointing North
	Y_DELTA_WORLD: REAL; // y delta in world frame (vs TD frame as given by gps)
	X_DELTA_WORLD: REAL; // not used here except to call function to get Y
END_VAR

// calculate how much we need to move bs by to align end (yaw pivot) with y of target 

GpsTdToWorldFixedYaw( X_TD_WP := X_TD_WP, Y_TD_WP := Y_TD_WP, YAW_BEGIN := HEADING_OFFSET_GPS, X_WORLD_WP => X_DELTA_WORLD, Y_WORLD_WP => Y_DELTA_WORLD);

BS_ANGLE_WORLD := YAW_ANGLE - HEADING_OFFSET_GPS;
BS_PIVOT_TO_YAW_PIVOT_Y_WORLD := SIN_DEG(BS_ANGLE_WORLD) * BS_LENGTH;
BS_PIVOT_TO_TARGET_Y_DELTA := BS_PIVOT_TO_YAW_PIVOT_Y_WORLD + Y_DELTA_WORLD;
IF ABS(BS_PIVOT_TO_TARGET_Y_DELTA) > BS_LENGTH THEN
	BS_PIVOT_TO_TARGET_Y_HEADING := BS_ANGLE_WORLD;
ELSE
	BS_PIVOT_TO_TARGET_Y_HEADING := ASIN_DEG( BS_PIVOT_TO_TARGET_Y_DELTA / BS_LENGTH );
END_IF

GPS_Y_TO_BS_ANGLE :=  BS_PIVOT_TO_TARGET_Y_HEADING - BS_ANGLE_WORLD ;

END_FUNCTION

// StandardPLC/Application/POUs/GPS/GpsAutoTrack
(* autotrack to gps target

create approach curve by floating target point that moves from 1/3 of distance to target
to 4 m behind target, then align to target and finish drive straignt on
*)
FUNCTION GpsAutoTrack : BOOL   // autotrack to gps target
VAR_INPUT
	// leave as input in case we want to control to a different point, eg 3rd leg motor
	X_OFFSET_BEGIN: REAL := 0; // offsets from WP given by gps, in TD frame, + is forward of operator 
	Y_OFFSET_BEGIN: REAL := 0; // + is to the right of operator (facing forward at rear [mast end] of TD)
	YAW_OFFSET_BEGIN: REAL := 0; // heading offset to rotate by as given by gps, + is moving mast to the right (CCW) of operator
	//Z_OFFSET_BEGIN: REAL := 0; // + is up;  if we want to add 3d functionality
END_VAR
VAR_OUTPUT
	LEFT_TRACK_OUTPUT_MAGNITUDE: INT := 0; // send as percent to joystick controller
	RIGHT_TRACK_OUTPUT_MAGNITUDE: INT := 0;
	LEFT_TRACK_OUTPUT_POSITIVE: BOOL := TRUE;
	RIGHT_TRACK_OUTPUT_POSITIVE: BOOL := TRUE;
END_VAR
VAR
	X_OFFSETS: ARRAY [1..9] OF REAL := [9(0)];
	Y_OFFSETS: ARRAY [1..9] OF REAL := [9(0)];
	YAW_OFFSETS: ARRAY [1..9] OF REAL := [9(0)];
	BS_ANGLE_NS_DELTA: REAL := 0;
	BS_ANGLE_WORLD_NS: REAL := 0;
	BS_ANGLE_NS_TO_Y_TARGET_DELTA: REAL := 0;
	YAW_ARM_LENGTH: REAL := 135; // 135 for TD3 with x slide at 0
	//HEADING_TO_TARGET: REAL := 0;
	HEADING_TO_TARGET_OFFSET: REAL := 0;

	
	//LEFT_TRACK_OUTPUT: REAL := 0;
	//RIGHT_TRACK_OUTPUT: REAL := 0;
	LEFT_TRACK_POSITIVE: BOOL := TRUE;
	RIGHT_TRACK_POSITIVE: BOOL := TRUE;
	PROXIMITY_SLOWING_FACTOR: REAL := 1;
	MANUAL_SPEED_REDUCING_FACTOR: REAL := 1;
	GPS_AUTO_TRACK_JOYSTICK_LIMIT: REAL := 70;
END_VAR


X_OFFSET_BEGIN := X_OFFSET_BEGIN/10; // convert mm to cm
Y_OFFSET_BEGIN := Y_OFFSET_BEGIN/10; // convert mm to cm
debug[30] := X_OFFSET_BEGIN;
debug[31] := Y_OFFSET_BEGIN;
//YAW_OFFSET_BEGIN := YAW_OFFSET_BEGIN; // deg to deg
//Z_OFFSET_BEGIN := Z_OFFSET_BEGIN/10; // convert mm to cm
YAW_ARM_LENGTH := YAW_PIVOT_TO_DRILL_ROD + AXES[AXIS_X_SLIDE].FEEDBACK.POSITION_ENGR;
//(* 
// * WP frame - origin at WP *
//  (if 3d have to first rotate at wp to get pitch and roll aligned with yaw arm)
// 1) translate origin to reference yaw pivot (translation)
(*
IF ABS(Y_OFFSET_BEGIN < 50) AND ABS(YAW_OFFSET_BEGIN) < 0.2 AND THEN
	HEADING_TO_TARGET := 0;
END_IF
*)

//YAW_OFFSET_BEGIN := YAW_OFFSET_BEGIN; // deg to deg
//Z_OFFSET_BEGIN := Z_OFFSET_BEGIN/10; // convert mm to cm

//(* 
// * WP frame - origin at WP *
//  (if 3d have to first rotate at wp to get pitch and roll aligned with yaw arm)
// 1) translate origin to reference yaw pivot (translation)

X_OFFSETS[1] := X_OFFSET_BEGIN - YAW_ARM_LENGTH;
Y_OFFSETS[1] := Y_OFFSET_BEGIN;

// * WP frame - origin at yaw pivot *
// 2) rotate origin at yaw pivot to match bs frame (rotation)
// YAW_ROTATION := AXES[AXIS_YAW].FEEDBACK.POSITION_ENGR; // offset from Boom Swing

X_OFFSETS[2] := X_OFFSETS[1] * COS_DEG(AXES[AXIS_YAW].FEEDBACK.POSITION_ENGR) - Y_OFFSETS[1] * SIN_DEG(AXES[AXIS_YAW].FEEDBACK.POSITION_ENGR); // rotate origin at yaw pivot by gps heading offset
Y_OFFSETS[2] := X_OFFSETS[1] * SIN_DEG(AXES[AXIS_YAW].FEEDBACK.POSITION_ENGR) + Y_OFFSETS[1] * COS_DEG(AXES[AXIS_YAW].FEEDBACK.POSITION_ENGR);

// * BS frame - origin AT yaw pivot *
// 3) translate origin to bs pivot

X_OFFSETS[3] := X_OFFSETS[2] - BS_PIVOT_TO_YAW_PIVOT;
Y_OFFSETS[3] := Y_OFFSETS[2];
debug[32] := X_OFFSETS[3];
debug[33] := Y_OFFSETS[3];

// * BS frame - origin at BS pivot *
// 4) rotate origin at bs pivot to world frame
//	- rotate by BS_ANGLE_NS_DELTA
BS_ANGLE_NS_DELTA := YAW_OFFSET_BEGIN + -1 * AXES[AXIS_YAW].FEEDBACK.POSITION_ENGR; //(Yaw is opposite sign)
BS_ANGLE_WORLD_NS := BS_ANGLE_NS_DELTA + AXES[AXIS_BOOM_SWING].FEEDBACK.POSITION_ENGR;

X_OFFSETS[4] := X_OFFSETS[3] * COS_DEG(BS_ANGLE_NS_DELTA) - Y_OFFSETS[3] * SIN_DEG(BS_ANGLE_NS_DELTA); // rotate origin at yaw pivot by gps heading offset
Y_OFFSETS[4] := X_OFFSETS[3] * SIN_DEG(BS_ANGLE_NS_DELTA) + Y_OFFSETS[3] * COS_DEG(BS_ANGLE_NS_DELTA);
debug[34] := X_OFFSETS[4];
debug[35] := Y_OFFSETS[4];

// * WORLD frame - origin at BS pivot *
IF ABS(X_OFFSETS[4]) > YAW_ARM_LENGTH + BS_PIVOT_TO_YAW_PIVOT THEN
	X_OFFSETS[5] := X_OFFSETS[4] / 5 ; // get ahead of 
	//Y_OFFSETS[5] := Y_OFFSETS[4];
	Y_OFFSETS[5] := Y_OFFSETS[4] * MIN(ABS(X_OFFSETS[4]) / 150, 1) ;

ELSE
	X_OFFSETS[5] := X_OFFSET_BEGIN; // get ahead of 
	Y_OFFSETS[5] := Y_OFFSETS[4];
END_IF

// translate target ccordinates to greater of 1/3 of remaining distance or 4 m
(*
IF X_OFFSETS[4] >= -420 THEN
	//(*
	IF X_OFFSETS[4] > 420 THEN
		X_OFFSETS[5] := MAX(( X_OFFSETS[4] / 4 ), 400); // get ahead of 
		(*
		X_OFFSETS[5] := X_OFFSETS[4] / 5 ; // get ahead of 
		Y_OFFSETS[5] := Y_OFFSETS[4] * ABS(X_OFFSETS[4]) / 400 ;
		//*)
	ELSE //*)
		X_OFFSETS[5] := X_OFFSETS[4] / 3;
		//Y_OFFSETS[5] := Y_OFFSETS[4];
	END_IF
ELSE
	IF X_OFFSETS[4] < -420 THEN
		//X_OFFSETS[5] := MIN(( X_OFFSETS[4] / 4 ), -400); // get ahead of 
		(*
		X_OFFSETS[5] := X_OFFSETS[4] / 5 ; // get ahead of 
		Y_OFFSETS[5] := Y_OFFSETS[4] * ABS(X_OFFSETS[4]) / 400 ; //*)
	ELSE
		X_OFFSETS[5] := X_OFFSETS[4] / 3;
		//Y_OFFSETS[5] := Y_OFFSETS[4];
	END_IF	
END_IF
*)

// OFFSESTS[5] are path target points in world frame from bs pivot13
debug[36] := X_OFFSETS[5];
debug[37] := Y_OFFSETS[5];
// get heading offset from North South line to new target
IF  X_OFFSETS[5] = 0 THEN // avoid /0 and keep approach orientation (+ x offset)
	 X_OFFSETS[5] := 0.1;
END_IF
IF ABS (X_OFFSETS[4] ) > 200 THEN // world frame x from bs pivot, eliminate divide by zero when close
	HEADING_TO_TARGET := ATAN_DEG ( - Y_OFFSETS[5] / X_OFFSETS[5] );
ELSE
	HEADING_TO_TARGET := 0;
END_IF

// get heading offset from machine heading
HEADING_TO_TARGET_OFFSET := YAW_OFFSET_BEGIN + HEADING_TO_TARGET;
debug[38] := HEADING_TO_TARGET_OFFSET;
// drive tracks to head to new target

 // reduce magnitude as approach target
PROXIMITY_SLOWING_FACTOR := MIN (ABS(X_OFFSET_BEGIN + 15)/200 , 1); // start slowing at 1m (offset already /10 above)
//PROXIMITY_SLOWING_FACTOR := MIN (ABS(X_OFFSETS[4] + 0.5)/10 , 1); // start slowing at 1m (offset already /10 above)
debug[39] := PROXIMITY_SLOWING_FACTOR;
//ROLL_SLOWING_FACTOR := MIN (xxxx ,1 ); // go slower if TD tilted sideways
//PITCH_SLOWING_FACTOR := MIN (xxxx ,1 ); // go slower if tilted up or down a hill
// let operator moderate speed with joysticks:
REMOTE.LJ_LR := 100;
REMOTE.RJ_LR := 100;
MANUAL_SPEED_REDUCING_FACTOR := MAX ( ( ((( ABS(REMOTE.LJ_LR) + ABS(REMOTE.RJ_LR) ) / 2 ) - GPS_AUTO_TRACK_JOYSTICK_LIMIT ) / ( 100 - GPS_AUTO_TRACK_JOYSTICK_LIMIT ) ) , 0 ); 

LEFT_TRACK_OUTPUT := MANUAL_SPEED_REDUCING_FACTOR * PROXIMITY_SLOWING_FACTOR * MAX ( MIN ( - HEADING_TO_TARGET_OFFSET * 1.5 + 90, 100), -100); // limit to -100 < x < 100
//LEFT_TRACK_OUTPUT := PROXIMITY_SLOWING_FACTOR * MAX ( MIN ( HEADING_TO_TARGET * 1.5 + 90, 100), -100); // limit to -100 < x < 100

debug[40] := LEFT_TRACK_OUTPUT;
IF LEFT_TRACK_OUTPUT < 0 THEN
	LEFT_TRACK_POSITIVE := FALSE;
ELSE
	LEFT_TRACK_POSITIVE := TRUE;
END_IF
RIGHT_TRACK_OUTPUT := MANUAL_SPEED_REDUCING_FACTOR * PROXIMITY_SLOWING_FACTOR * MAX ( MIN ( HEADING_TO_TARGET_OFFSET * 1.5 + 90, 100), -100);// limit to 100
//RIGHT_TRACK_OUTPUT := PROXIMITY_SLOWING_FACTOR * MAX ( MIN ( - HEADING_TO_TARGET * 1.5 + 90, 100), -100);// limit to 100

debug[41] := RIGHT_TRACK_OUTPUT;
IF RIGHT_TRACK_OUTPUT < 0 THEN
	RIGHT_TRACK_POSITIVE := FALSE;
ELSE
	RIGHT_TRACK_POSITIVE := TRUE;
END_IF

IF X_OFFSETS[5] >= 0 THEN // going forward, normal situation
	LEFT_TRACK_OUTPUT_MAGNITUDE:= TO_INT ( ABS( LEFT_TRACK_OUTPUT) );  // max 100
	LEFT_TRACK_OUTPUT_POSITIVE := NOT LEFT_TRACK_POSITIVE; // tracks are positive to move backward and vice versa
	RIGHT_TRACK_OUTPUT_MAGNITUDE:= TO_INT ( ABS( RIGHT_TRACK_OUTPUT ) );  // max 100
	RIGHT_TRACK_OUTPUT_POSITIVE:= NOT RIGHT_TRACK_POSITIVE;
ELSE // swap directions
	RIGHT_TRACK_OUTPUT_MAGNITUDE:= TO_INT ( ABS( LEFT_TRACK_OUTPUT ) );  // max 100
	RIGHT_TRACK_OUTPUT_POSITIVE := (LEFT_TRACK_POSITIVE);
	LEFT_TRACK_OUTPUT_MAGNITUDE := TO_INT ( ABS( RIGHT_TRACK_OUTPUT ) );  // max 100
	LEFT_TRACK_OUTPUT_POSITIVE := (RIGHT_TRACK_POSITIVE);
 END_IF

 (*
IF X_OFFSETS[5] >= 0 THEN
	AXES[AXIS_TRACK_LEFT].OUTPUT.MAGNITUDE := TO_WORD( ABS( LEFT_TRACK_OUTPUT ) * 10);  // max 1000
	AXES[AXIS_TRACK_LEFT].OUTPUT.POSITIVE := LEFT_TRACK_POSITIVE;
	AXES[AXIS_TRACK_RIGHT].OUTPUT.MAGNITUDE := TO_WORD( ABS( RIGHT_TRACK_OUTPUT ) * 10);  // max 1000
	AXES[AXIS_TRACK_RIGHT].OUTPUT.POSITIVE := RIGHT_TRACK_POSITIVE;
ELSE
	AXES[AXIS_TRACK_RIGHT].OUTPUT.MAGNITUDE := TO_WORD( ABS( LEFT_TRACK_OUTPUT ) * 10);  // max 1000
	AXES[AXIS_TRACK_RIGHT].OUTPUT.POSITIVE := NOT(LEFT_TRACK_POSITIVE);
	AXES[AXIS_TRACK_LEFT].OUTPUT.MAGNITUDE := TO_WORD( ABS( RIGHT_TRACK_OUTPUT ) * 10);  // max 1000
	AXES[AXIS_TRACK_LEFT].OUTPUT.POSITIVE := NOT(RIGHT_TRACK_POSITIVE);
 END_IF
*)

END_FUNCTION

// StandardPLC/Application/POUs/Utilities/Conversions/ATAN_DEG
FUNCTION ATAN_DEG: REAL
VAR_INPUT
	VALUE: REAL;
END_VAR
VAR
END_VAR

ATAN_DEG := (180 * ATAN(VALUE)) / 3.14159;

END_FUNCTION

// StandardPLC/Application/POUs/Test_PRGs/Parsing
PROGRAM Parsing
VAR
	Reals: ARRAY [1..20] OF REAL := [20(0)]; //9223372036854775808;
	TEST_BOOLS: ARRAY [1..20] OF BOOL := [20(0)];	
	LWords: ARRAY [1..20] OF LWORD := [20(0)];
END_VAR


Reals[1] := 9223372036854775808;
Lwords[1] := TO_LWORD(Reals[1]);

TEST_BOOLS[1] := TO_BOOL(SHR(LWords[1], 63));

Reals[2] := 6.5432;
Reals[3] := Reals[2] + 0.00001;
Lwords[2] := TO_LWORD(Reals[2]);// rounds to non decimal
Lwords[3] := TO_LWORD(Reals[3]);
//TEST_BOOLS[2] := TO_BOOL(SHR(Reals[1], 63)); // has to be non-decimal

END_PROGRAM

// StandardPLC/Application/POUs/Test_PRGs/pnezD_decoding
PROGRAM pnezD_decoding
VAR
	// *****function vars*****
	CODE_START: INT :=0;
	
	// *****sim vars*****
	D_LENGTH: USINT := 0;
	init: BOOL := TRUE;
	CHARS: ARRAY [1..50] OF STRING(1);
	PARAMETERS: ARRAY [1..50] OF STRING(5);
	T_TYPE: STRING := '';
	Test: REAL;
	VALID: BOOL := FALSE;
	
	TRUSS_CODES: ARRAY [0..2, 1..2] OF STRING(1) := ['i','I','c','C','e','E'];
	letter_index : USINT := 1;
	case_index: USINT := 0;
	dbug: ARRAY [1..40] OF USINT := [40(0)];
	
	pnezDlast: STRING(64) := '';
	file_index: USINT := 0;
END_VAR

//  set up test parameters
IF init THEN
	init := FALSE;
	//GPS_PNEZD_D := 'Test: J+0020020ZZ1075070C end';
	//GPS_PNEZD_D := 'test: J-1122233445556677I end';
	//GPS_PNEZD_D := 'Test: J+1122233445556677E end';
	//GPS_PNEZD_D := 'Testj-: J-1122233ZZ555zzZZI end';
	GPS_PNEZD_D := 'TestJ: J-0020020ZZ1225070C end';
	VALID := DecodePnezD();
END_IF


// run function
IF GPS_PNEZD_D <> pnezDlast THEN
	pnezDlast := GPS_PNEZD_D;
	
	//run function
	VALID := DecodePnezD();
	SCREW_PARAMS_CUSTOM[file_index] := SCREW_PARAMS_CUSTOM[0];
	file_index := MIN(file_index + 1, 10);
	//test enum
	IF SCREW_PARAMETERS[TRUSS_TYPE] = 1 THEN
		T_TYPE := 'Center';
	ELSIF SCREW_PARAMETERS[TRUSS_TYPE] = 0 THEN
		T_TYPE := 'Interior';
	ELSIF SCREW_PARAMETERS[TRUSS_TYPE] = 2 THEN
		T_TYPE := 'Exterior';
	ELSE 
		T_TYPE := 'NA';
	END_IF
	
	(* see iteration
	//
	VALID := TRUE; 
	// Find the J_code
	CODE_START := FIND(GPS_PNEZD_D,'J+') + FIND(GPS_PNEZD_D,'J-');
	IF (CODE_START = 0) THEN
		VALID := FALSE; // did not find a valid code
		dbug[1] := dbug[1] + 1;
		RETURN;
	ELSE
		VALID := FALSE;
		FOR letter_index := 0 TO 2 DO
			dbug[2] := dbug[2] + 1;
			FOR case_index := 1 TO 2 DO
				dbug[3] := dbug[3] + 1;
				IF MID(GPS_PNEZD_D, 1, CODE_START + 18) = TRUSS_CODES[letter_index, case_index] THEN 
					VALID := TRUE;
					SCREW_PARAMETERS[TRUSS_TYPE] := TO_REAL(letter_index);
					dbug[4] := dbug[4] + 1;
				END_IF
				
			END_FOR
		END_FOR
		IF VALID = FALSE THEN
			dbug[5] := dbug[5] + 1;
			RETURN;
		END_IF
	END_IF
		dbug[6] := dbug[6] + 1;
		CODE_START := CODE_START + 1;
		// pull out the parameters
		SCREW_PARAMETERS[NS_PITCH] := STRING_TO_REAL(MID(GPS_PNEZD_D, 3, CODE_START));
		CODE_START := CODE_START + 3;
		SCREW_PARAMETERS[SCREW_LENGTH] := STRING_TO_REAL(MID(GPS_PNEZD_D, 3, CODE_START));
		CODE_START := CODE_START + 3;
		SCREW_PARAMETERS[TRUSS_VERT_ANGLE] := STRING_TO_REAL(MID(GPS_PNEZD_D, 2, CODE_START));
		CODE_START := CODE_START + 2;
		IF MID(GPS_PNEZD_D, 2, CODE_START) = 'ZZ' OR MID(GPS_PNEZD_D, 2, CODE_START) = 'zz' THEN
			SCREW_PARAMETERS[THIRD_LEG_VERT_ANGLE] := NA;
		ELSE
			SCREW_PARAMETERS[THIRD_LEG_VERT_ANGLE] := STRING_TO_REAL(MID(GPS_PNEZD_D, 2, CODE_START));
		END_IF
		CODE_START := CODE_START + 2;
		SCREW_PARAMETERS[EMBED_LENGTH] := STRING_TO_REAL(MID(GPS_PNEZD_D, 3, CODE_START));
		CODE_START := CODE_START + 3;
		IF MID(GPS_PNEZD_D, 2, CODE_START) = 'ZZ' OR MID(GPS_PNEZD_D, 2, CODE_START) = 'zz' THEN
			SCREW_PARAMETERS[IE_MIN_HAMMER] := NA;
		ELSE
			SCREW_PARAMETERS[IE_MIN_HAMMER] := STRING_TO_REAL(MID(GPS_PNEZD_D, 2, CODE_START));
		END_IF
		CODE_START := CODE_START + 2;
		IF MID(GPS_PNEZD_D, 2, CODE_START) = 'ZZ' OR MID(GPS_PNEZD_D, 2, CODE_START) = 'zz' THEN
			SCREW_PARAMETERS[IE_MIN_EMBED] := NA;
		ELSE
			SCREW_PARAMETERS[IE_MIN_EMBED] := STRING_TO_REAL(MID(GPS_PNEZD_D, 2, CODE_START));
		END_IF
		CODE_START := CODE_START + 2;
		//*)
END_IF
//VALID := DecodePnezD();



//FOR i := 1 TO LEN(GPS_PNEZD_D) DO

END_PROGRAM

// StandardPLC/Application/POUs/GPS/DecodePnezD
FUNCTION DecodePnezD : BOOL
VAR_INPUT
END_VAR
VAR
	CODE_START: INT :=0;
	PARAMETERS: ARRAY [1..3] OF STRING(2);
	TRUSS_CODES: ARRAY [0..2, 1..2] OF STRING(1) := ['i','I','c','C','e','E'];
	letter_index : USINT := 1;
	case_index: USINT := 0;
END_VAR

//
DecodePnezD := TRUE; 
// Find the J_code
CODE_START := FIND(GPS_PNEZD_D,'J+') + FIND(GPS_PNEZD_D,'J-');
IF (CODE_START = 0) THEN
	DecodePnezD := FALSE; // did not find a valid code
	RETURN;
ELSE
	DecodePnezD := FALSE;
	FOR letter_index := 0 TO 2 DO
		FOR case_index := 1 TO 2 DO
			IF MID(GPS_PNEZD_D, 1, CODE_START + 18) = TRUSS_CODES[letter_index, case_index] THEN 
				DecodePnezD := TRUE;
				SCREW_PARAMETERS[TRUSS_TYPE] := TO_REAL(letter_index);
				SCREW_PARAMS_CUSTOM[0].TRUSS_TYPE := TO_USINT(letter_index);
			END_IF
			
		END_FOR
	END_FOR
	IF DecodePnezD = FALSE THEN
		RETURN;
	END_IF
END_IF
	
